# B&R Automation Studio project TD52 (part 61)

```c
  /* Logic: '<S427>/Logical Operator11' incorporates:
   *  Logic: '<S427>/Logical Operator25'
   *  UnitDelay: '<S427>/Unit Delay4'
   */
  rtb_LogicalOperator_in = ((!Gen2_ref_DWork->TOF_state) &&
    rtb_LogicalOperator5_mv && rtb_dbg_HLCi &&
    Gen2_ref_B->BusInput3.LR.bP_LoadReject_Active && rtb_RelationalOperator2_j);

  /* Sum: '<S427>/Sum6' incorporates:
   *  Constant: '<S427>/Constant7'
   *  Gain: '<S427>/Gain3'
   */
  rtb_Divide4_ia = 0.001 * Gen2_ref_B->BusInput3.LR.rTi_LR_GasStop + 0.01;

  /* Outputs for Atomic SubSystem: '<S427>/TOF1' */
  Gen2_ref_TOF(rtb_LogicalOperator_in, rtb_Divide4_ia, &Gen2_ref_B->TOF1_o,
               &Gen2_ref_DWork->TOF1_o, inst);

  /* End of Outputs for SubSystem: '<S427>/TOF1' */

  /* Outputs for Atomic SubSystem: '<S427>/TP' */
  Gen2_ref_TP(rtb_LogicalOperator_in, rtb_Divide4_ia, &Gen2_ref_B->TP_p,
              &Gen2_ref_DWork->TP_p, inst);

  /* End of Outputs for SubSystem: '<S427>/TP' */

  /* Switch: '<S427>/Switch1' */
  if (Gen2_ref_B->BusInput3.LR.bTiTOF_GasSTop) {
    rtb_TOF_IN = Gen2_ref_B->TOF1_o.LogicalOperator1;
  } else {
    rtb_TOF_IN = Gen2_ref_B->TP_p.LogicalOperator1;
  }

  /* End of Switch: '<S427>/Switch1' */

  /* Switch: '<Root>/GasStop1' */
  rtb_dbg_HLCi = ((!rtb_LogicalOperator) && rtb_TOF_IN);

  /* Outputs for Atomic SubSystem: '<S8>/BDC_Trajectory' */
  /* Gain: '<S345>/Gain8' incorporates:
   *  Gain: '<S417>/Gain8'
   *  Gain: '<S760>/Gain8'
   */
  rtb_Switch_ct_tmp = 100000.0 * Gen2_ref_B->BusInput3.traj.rPr_p2s_Sr_Man;

  /* Product: '<S413>/delta rise limit' incorporates:
   *  Gain: '<S345>/Gain8'
   *  Product: '<S434>/delta rise limit'
   *  Product: '<S795>/delta rise limit'
   *  SampleTimeMath: '<S413>/sample time'
   *
   * About '<S413>/sample time':
   *  y = K where K = ( w * Ts )
   */
  rtb_Divide_mr_tmp_0 = rtb_Switch_ct_tmp * 0.01;

  /* End of Outputs for SubSystem: '<S8>/BDC_Trajectory' */
  rtb_Divide_kp = rtb_Divide_mr_tmp_0;

  /* Gain: '<S4>/bar2Pa6' incorporates:
   *  DataTypeConversion: '<S4>/Data Type Conversion27'
   */
  rtb_bar2Pa6 = 100000.0 * Gen2_ref_B->BusInput.rPr_p2sMan;

  /* Logic: '<S4>/Logical Operator3' incorporates:
   *  Logic: '<S4>/Logical Operator2'
   */
  rtb_LogicalOperator_in = ((!rtb_LogicalOperator) || rtb_bResetBdc);

  /* DiscreteIntegrator: '<S345>/Discrete-Time Integrator' */
  if (rtb_LogicalOperator_in || (Gen2_ref_DWork->DiscreteTimeIntegrator_PrevRese
       != 0)) {
    Gen2_ref_DWork->DiscreteTimeIntegrator_DSTATE = 1.0;
  }

  if (Gen2_ref_DWork->DiscreteTimeIntegrator_DSTATE >= 1.0) {
    Gen2_ref_DWork->DiscreteTimeIntegrator_DSTATE = 1.0;
  } else if (Gen2_ref_DWork->DiscreteTimeIntegrator_DSTATE <= 0.0) {
    Gen2_ref_DWork->DiscreteTimeIntegrator_DSTATE = 0.0;
  }

  /* Logic: '<S345>/Logical Operator' incorporates:
   *  Constant: '<S345>/Constant2'
   *  DiscreteIntegrator: '<S345>/Discrete-Time Integrator'
   *  RelationalOperator: '<S345>/Relational Operator'
   */
  rtb_LogicalOperator_cn = ((0.99 <=
    Gen2_ref_DWork->DiscreteTimeIntegrator_DSTATE) || rtb_LogicalOperator_in);

  /* Delay: '<S413>/Delay' */
  Gen2_ref_DWork->icLoad_n = ((((Gen2_ref_PrevZCSigState->Delay_Reset_ZCE_k == 1)
    != (int32_T)rtb_LogicalOperator_cn) &&
    (Gen2_ref_PrevZCSigState->Delay_Reset_ZCE_k != 3)) || rtb_LogicalOperator_cn
    || Gen2_ref_DWork->icLoad_n);
  Gen2_ref_PrevZCSigState->Delay_Reset_ZCE_k = rtb_LogicalOperator_cn;
  if (Gen2_ref_DWork->icLoad_n) {
    Gen2_ref_DWork->Delay_DSTATE_n = rtb_bar2Pa6;
  }

  /* Sum: '<S413>/Difference Inputs1' incorporates:
   *  Delay: '<S413>/Delay'
   *  Switch: '<S413>/etaVolConst'
   */
  rtb_Divide4_ia = rtb_bar2Pa6 - Gen2_ref_DWork->Delay_DSTATE_n;

  /* Switch: '<S416>/Switch2' incorporates:
   *  Product: '<S413>/delta rise limit'
   *  RelationalOperator: '<S416>/LowerRelop1'
   */
  if (!(rtb_Divide4_ia > rtb_Divide_mr_tmp_0)) {
    /* Product: '<S413>/delta fall limit' incorporates:
     *  Gain: '<S345>/Gain15'
     *  Gain: '<S345>/Gain8'
     *  SampleTimeMath: '<S413>/sample time'
     *
     * About '<S413>/sample time':
     *  y = K where K = ( w * Ts )
     */
    rtb_Switch_ed = -rtb_Switch_ct_tmp * 0.01;

    /* Switch: '<S416>/Switch' incorporates:
     *  RelationalOperator: '<S416>/UpperRelop'
     */
    if (rtb_Divide4_ia < rtb_Switch_ed) {
      rtb_Divide_kp = rtb_Switch_ed;
    } else {
      rtb_Divide_kp = rtb_Divide4_ia;
    }

    /* End of Switch: '<S416>/Switch' */
  }

  /* End of Switch: '<S416>/Switch2' */

  /* Sum: '<S413>/Difference Inputs2' incorporates:
   *  Delay: '<S413>/Delay'
   */
  rtb_Divide4_ia = rtb_Divide_kp + Gen2_ref_DWork->Delay_DSTATE_n;

  /* Outputs for Atomic SubSystem: '<S345>/p2sfilt' */
  Gen2_ref_N_TC_HP_filt(rtb_Divide4_ia,
                        Gen2_ref_B->BusInput3.traj.rTiF_Pr_p2s_Man,
                        rtb_LogicalOperator_cn, &Gen2_ref_B->p2sfilt,
                        &Gen2_ref_DWork->p2sfilt, inst);

  /* End of Outputs for SubSystem: '<S345>/p2sfilt' */

  /* Gain: '<S875>/kW2W1' incorporates:
   *  Gain: '<S343>/Pa2bar2'
   *  Gain: '<S344>/kW2W1'
   *  Gain: '<S586>/Gain1'
   *  Gain: '<S639>/kW2W'
   *  Gain: '<S761>/kW2W'
   *  Switch: '<S761>/Switch2'
   */
  rtb_Product1_aq = 1000.0 * Gen2_ref_B->BusInput3.eng.rP_Nom;

  /* Product: '<S881>/delta rise limit' incorporates:
   *  Gain: '<S875>/kW2W1'
   *  Product: '<S875>/Divide1'
   *  SampleTimeMath: '<S881>/sample time'
   *
   * About '<S881>/sample time':
   *  y = K where K = ( w * Ts )
   */
  rtb_Divide2_a = rtb_Product1_aq *
    Gen2_ref_B->BusInput3.traj.rP_Ramp_IncGrad_Norm * 0.01;

  /* Product: '<S875>/Product' incorporates:
   *  Gain: '<S875>/kW2W1'
   */
  rtb_Product_gj = rtb_Product1_aq * Gen2_ref_B->BusInput3.eng.rP_Start_Norm;

  /* Outputs for Atomic SubSystem: '<S194>/Pel_filt' */
  Gen2_ref_N_TC_HP_filt(rtb_Gain2_ao, Gen2_ref_B->BusInput3.inFilt.rTiF_P,
                        rtb_bResetBdc, &Gen2_ref_B->Pel_filt,
                        &Gen2_ref_DWork->Pel_filt, inst);

  /* End of Outputs for SubSystem: '<S194>/Pel_filt' */

  /* MATLAB Function: '<S874>/MATLAB Function' */
  if (!Gen2_ref_B->BusInput.tLvrt.bLvrtFlg) {
    rtb_PactOut = Gen2_ref_B->Pel_filt.Switch;
    rtb_PrefOut = rtb_kW2W;
    Gen2_ref_DWork->LVRTFlgRise = false;
  } else if (Gen2_ref_B->BusInput.tLvrt.bLvrtFlg &&
             (!Gen2_ref_DWork->LVRTFlgRise)) {
    Gen2_ref_DWork->PFix = Gen2_ref_B->Pel_filt.Switch;
    rtb_PactOut = Gen2_ref_DWork->PFix;
    rtb_PrefOut = Gen2_ref_DWork->PFix;
    Gen2_ref_DWork->LVRTFlgRise = true;
  } else {
    rtb_PactOut = Gen2_ref_DWork->PFix;
    rtb_PrefOut = Gen2_ref_DWork->PFix;
  }

  /* End of MATLAB Function: '<S874>/MATLAB Function' */

  /* Switch: '<S881>/etaVolConst' incorporates:
   *  Constant: '<S875>/ tde2'
   *  Gain: '<S875>/kW2W1'
   *  RelationalOperator: '<S878>/LowerRelop1'
   *  RelationalOperator: '<S878>/UpperRelop'
   *  Switch: '<S878>/Switch'
   *  Switch: '<S878>/Switch2'
   */
  if (Gen2_ref_B->BusInput.bResetTraj) {
    rtb_PactOut = rtb_Product_gj;
  } else {
    if (rtb_PrefOut > rtb_Product1_aq) {
      /* Switch: '<S878>/Switch2' incorporates:
       *  Gain: '<S875>/kW2W1'
       */
      rtb_PrefOut = rtb_Product1_aq;
    } else if (rtb_PrefOut < 1.0) {
      /* Switch: '<S878>/Switch' incorporates:
       *  Constant: '<S875>/ tde2'
       *  Switch: '<S878>/Switch2'
       */
      rtb_PrefOut = 1.0;
    }

    /* Switch: '<S880>/Switch2' incorporates:
     *  Constant: '<S875>/ tde2'
     *  Gain: '<S875>/kW2W1'
     *  RelationalOperator: '<S878>/UpperRelop'
     *  RelationalOperator: '<S880>/LowerRelop1'
     *  RelationalOperator: '<S880>/UpperRelop'
     *  Switch: '<S878>/Switch'
     *  Switch: '<S878>/Switch2'
     *  Switch: '<S880>/Switch'
     */
    if (rtb_PactOut > rtb_Product1_aq) {
      rtb_PactOut = rtb_Product1_aq;
    } else if (rtb_PactOut < rtb_Product_gj) {
      /* Switch: '<S880>/Switch' */
      rtb_PactOut = rtb_Product_gj;
    }

    /* End of Switch: '<S880>/Switch2' */

    /* Sum: '<S875>/Sum10' incorporates:
     *  Gain: '<S875>/kW2W1'
     *  Product: '<S875>/Divide5'
     */
    rtb_PactOut += Gen2_ref_B->BusInput3.traj.rP_Diff_Max_Norm * rtb_Product1_aq;

    /* Switch: '<S879>/Switch2' incorporates:
     *  RelationalOperator: '<S879>/LowerRelop1'
     */
    if (!(rtb_PrefOut > rtb_PactOut)) {
      /* Switch: '<S879>/Switch' incorporates:
       *  Constant: '<S875>/ tde3'
       *  RelationalOperator: '<S879>/UpperRelop'
       */
      if (rtb_PrefOut < 1.0) {
        rtb_PactOut = 1.0;
      } else {
        rtb_PactOut = rtb_PrefOut;
      }

      /* End of Switch: '<S879>/Switch' */
    }

    /* End of Switch: '<S879>/Switch2' */
  }

  /* End of Switch: '<S881>/etaVolConst' */

  /* Delay: '<S881>/Delay' */
  Gen2_ref_DWork->icLoad_m = ((((Gen2_ref_PrevZCSigState->Delay_Reset_ZCE_b == 1)
    != (int32_T)Gen2_ref_B->BusInput.bResetTraj) &&
    (Gen2_ref_PrevZCSigState->Delay_Reset_ZCE_b != 3)) ||
    Gen2_ref_B->BusInput.bResetTraj || Gen2_ref_DWork->icLoad_m);
  Gen2_ref_PrevZCSigState->Delay_Reset_ZCE_b = Gen2_ref_B->BusInput.bResetTraj;
  if (Gen2_ref_DWork->icLoad_m) {
    Gen2_ref_DWork->Delay_DSTATE_oh = rtb_Product_gj;
  }

  /* Sum: '<S881>/Difference Inputs1' incorporates:
   *  Delay: '<S881>/Delay'
   */
  rtb_PactOut -= Gen2_ref_DWork->Delay_DSTATE_oh;

  /* Switch: '<S884>/Switch2' incorporates:
   *  RelationalOperator: '<S884>/LowerRelop1'
   */
  if (!(rtb_PactOut > rtb_Divide2_a)) {
    /* Product: '<S881>/delta fall limit' incorporates:
     *  Abs: '<S875>/Abs2'
     *  Gain: '<S875>/Gain2'
     *  Gain: '<S875>/kW2W1'
     *  Product: '<S875>/Divide2'
     *  SampleTimeMath: '<S881>/sample time'
     *
     * About '<S881>/sample time':
     *  y = K where K = ( w * Ts )
     */
    rtb_Switch_ed = -fabs(rtb_Product1_aq *
                          Gen2_ref_B->BusInput3.traj.rP_Ramp_DecGrad_Norm) *
      0.01;

    /* Switch: '<S884>/Switch' incorporates:
     *  RelationalOperator: '<S884>/UpperRelop'
     */
    if (rtb_PactOut < rtb_Switch_ed) {
      rtb_Divide2_a = rtb_Switch_ed;
    } else {
      rtb_Divide2_a = rtb_PactOut;
    }

    /* End of Switch: '<S884>/Switch' */
  }

  /* End of Switch: '<S884>/Switch2' */

  /* Sum: '<S881>/Difference Inputs2' incorporates:
   *  Delay: '<S881>/Delay'
   */
  rtb_Switch_ed = rtb_Divide2_a + Gen2_ref_DWork->Delay_DSTATE_oh;

  /* Outputs for Atomic SubSystem: '<S875>/Pd_filt' */
  Gen2_ref_Pd_filt(rtb_Switch_ed, Gen2_ref_B->BusInput3.traj.rTiFpowtraj,
                   rtb_Product_gj, Gen2_ref_B->BusInput.bResetTraj,
                   &Gen2_ref_B->Pd_filt_p, &Gen2_ref_DWork->Pd_filt_p, inst);

  /* End of Outputs for SubSystem: '<S875>/Pd_filt' */

  /* Gain: '<S344>/kW2W1' */
  rtb_kW2W1_h = rtb_Product1_aq;

  /* Product: '<S404>/delta rise limit' incorporates:
   *  Product: '<S344>/Divide1'
   *  SampleTimeMath: '<S404>/sample time'
   *
   * About '<S404>/sample time':
   *  y = K where K = ( w * Ts )
   */
  rtb_Divide2_a = rtb_kW2W1_h * Gen2_ref_B->BusInput3.traj.rP_Ramp_IncGrad_Norm *
    0.01;

  /* Product: '<S344>/Product' */
  rtb_PactOut = rtb_kW2W1_h * Gen2_ref_B->BusInput3.eng.rP_Start_Norm;

  /* Logic: '<Root>/Logical Operator1' incorporates:
   *  Logic: '<Root>/Logical Operator2'
   */
  rtb_LogicalOperator1_e = (Gen2_ref_B->BusInput.tLvrt.bLvrtFlg &&
    (!rtb_LogicalOperator_in));

  /* MATLAB Function: '<S339>/MATLAB Function' */
  if (!rtb_LogicalOperator1_e) {
    rtb_PactOut_o = Gen2_ref_B->Pel_filt.Switch;
    rtb_Product_gj = rtb_kW2W;
    Gen2_ref_DWork->LVRTFlgRise_e = false;
  } else if (!Gen2_ref_DWork->LVRTFlgRise_e) {
    Gen2_ref_DWork->PFix_g = Gen2_ref_B->Pel_filt.Switch;
    rtb_PactOut_o = Gen2_ref_DWork->PFix_g;
    rtb_Product_gj = Gen2_ref_DWork->PFix_g;
    Gen2_ref_DWork->LVRTFlgRise_e = true;
  } else {
    rtb_PactOut_o = Gen2_ref_DWork->PFix_g;
    rtb_Product_gj = Gen2_ref_DWork->PFix_g;
  }

  /* End of MATLAB Function: '<S339>/MATLAB Function' */

  /* Switch: '<S397>/Switch2' incorporates:
   *  Constant: '<S344>/ tde2'
   *  RelationalOperator: '<S397>/LowerRelop1'
   *  RelationalOperator: '<S397>/UpperRelop'
   *  Switch: '<S397>/Switch'
   */
  if (rtb_Product_gj > rtb_kW2W1_h) {
    rtb_PrefOut = rtb_kW2W1_h;
  } else if (rtb_Product_gj < 1.0) {
    /* Switch: '<S397>/Switch' incorporates:
     *  Constant: '<S344>/ tde2'
     */
    rtb_PrefOut = 1.0;
  } else {
    rtb_PrefOut = rtb_Product_gj;
  }

  /* End of Switch: '<S397>/Switch2' */

  /* Switch: '<S404>/etaVolConst' incorporates:
   *  RelationalOperator: '<S399>/LowerRelop1'
   *  RelationalOperator: '<S399>/UpperRelop'
   *  Switch: '<S399>/Switch'
   *  Switch: '<S399>/Switch2'
   */
  if (rtb_LogicalOperator_in) {
    rtb_Product_gj = rtb_PactOut;
  } else {
    if (rtb_PactOut_o > rtb_kW2W1_h) {
      /* Switch: '<S399>/Switch2' */
      rtb_Divide_kp = rtb_kW2W1_h;
    } else if (rtb_PactOut_o < rtb_PactOut) {
      /* Switch: '<S399>/Switch' incorporates:
       *  Switch: '<S399>/Switch2'
       */
      rtb_Divide_kp = rtb_PactOut;
    } else {
      /* Switch: '<S399>/Switch2' incorporates:
       *  Switch: '<S399>/Switch'
       */
      rtb_Divide_kp = rtb_PactOut_o;
    }

    /* Sum: '<S344>/Sum10' incorporates:
     *  Product: '<S344>/Divide5'
     *  RelationalOperator: '<S399>/UpperRelop'
     *  Switch: '<S399>/Switch'
     *  Switch: '<S399>/Switch2'
     */
    rtb_Product_gj = Gen2_ref_B->BusInput3.traj.rP_Diff_Max_Norm * rtb_kW2W1_h +
      rtb_Divide_kp;

    /* Switch: '<S398>/Switch2' incorporates:
     *  RelationalOperator: '<S398>/LowerRelop1'
     */
    if (!(rtb_PrefOut > rtb_Product_gj)) {
      /* Switch: '<S398>/Switch' incorporates:
       *  Constant: '<S344>/ tde3'
       *  RelationalOperator: '<S398>/UpperRelop'
       */
      if (rtb_PrefOut < 1.0) {
        rtb_Product_gj = 1.0;
      } else {
        rtb_Product_gj = rtb_PrefOut;
      }

      /* End of Switch: '<S398>/Switch' */
    }

    /* End of Switch: '<S398>/Switch2' */
  }

  /* End of Switch: '<S404>/etaVolConst' */

  /* Delay: '<S404>/Delay' */
  Gen2_ref_DWork->icLoad_k = ((((Gen2_ref_PrevZCSigState->Delay_Reset_ZCE_n == 1)
    != (int32_T)rtb_LogicalOperator_in) &&
    (Gen2_ref_PrevZCSigState->Delay_Reset_ZCE_n != 3)) || rtb_LogicalOperator_in
    || Gen2_ref_DWork->icLoad_k);
  Gen2_ref_PrevZCSigState->Delay_Reset_ZCE_n = rtb_LogicalOperator_in;
  if (Gen2_ref_DWork->icLoad_k) {
    Gen2_ref_DWork->Delay_DSTATE_g = rtb_PactOut;
  }

  /* Sum: '<S404>/Difference Inputs1' incorporates:
   *  Delay: '<S404>/Delay'
   */
  rtb_Product_gj -= Gen2_ref_DWork->Delay_DSTATE_g;

  /* Switch: '<S411>/Switch2' incorporates:
   *  RelationalOperator: '<S411>/LowerRelop1'
   */
  if (!(rtb_Product_gj > rtb_Divide2_a)) {
    /* Product: '<S404>/delta fall limit' incorporates:
     *  Abs: '<S344>/Abs2'
     *  Gain: '<S344>/Gain2'
     *  Product: '<S344>/Divide2'
     *  SampleTimeMath: '<S404>/sample time'
     *
     * About '<S404>/sample time':
     *  y = K where K = ( w * Ts )
     */
    rtb_deltafalllimit_ca = -fabs(rtb_kW2W1_h *
      Gen2_ref_B->BusInput3.traj.rP_Ramp_DecGrad_Norm) * 0.01;

    /* Switch: '<S411>/Switch' incorporates:
     *  RelationalOperator: '<S411>/UpperRelop'
     */
    if (rtb_Product_gj < rtb_deltafalllimit_ca) {
      rtb_Divide2_a = rtb_deltafalllimit_ca;
    } else {
      rtb_Divide2_a = rtb_Product_gj;
    }

    /* End of Switch: '<S411>/Switch' */
  }

  /* End of Switch: '<S411>/Switch2' */

  /* Sum: '<S404>/Difference Inputs2' incorporates:
   *  Delay: '<S404>/Delay'
   */
  rtb_Product_gj = rtb_Divide2_a + Gen2_ref_DWork->Delay_DSTATE_g;

  /* Outputs for Atomic SubSystem: '<S344>/Pd_filt' */
  Gen2_ref_Pd_filt(rtb_Product_gj, Gen2_ref_B->BusInput3.traj.rTiFpowtraj,
                   rtb_PactOut, rtb_LogicalOperator_in, &Gen2_ref_B->Pd_filt,
                   &Gen2_ref_DWork->Pd_filt, inst);

  /* End of Outputs for SubSystem: '<S344>/Pd_filt' */

  /* Gain: '<S344>/kW2W2' */
  rtb_PactOut = 1000.0 * rtb_kW2W1_h;

  /* Gain: '<S344>/kW2W3' */
  rtb_Divide2_a = 0.1 * rtb_PactOut;

  /* Outputs for Atomic SubSystem: '<S344>/WO1' */
  Gen2_ref_Filter1(rtb_PrefOut, Gen2_ref_B->BusInput3.traj.rTi_FSM_WO_1,
                   rtb_LogicalOperator_in, &Gen2_ref_B->WO1,
                   &Gen2_ref_DWork->WO1, inst);

  /* End of Outputs for SubSystem: '<S344>/WO1' */

  /* Outputs for Atomic SubSystem: '<S344>/WO2' */
  Gen2_ref_Filter3(Gen2_ref_B->WO1.Switch1,
                   Gen2_ref_B->BusInput3.traj.rTi_FSM_WO_2, Gen2_ref_ConstB.tde1,
                   rtb_LogicalOperator_in, &Gen2_ref_B->WO2,
                   &Gen2_ref_DWork->WO2, inst);

  /* End of Outputs for SubSystem: '<S344>/WO2' */

  /* Product: '<S344>/Divide3' */
  rtb_PrefOut = Gen2_ref_B->BusInput3.traj.rK_FSM_WO * Gen2_ref_B->WO2.Switch;

  /* Switch: '<S400>/Switch2' incorporates:
   *  RelationalOperator: '<S400>/LowerRelop1'
   */
  if (rtb_PrefOut > rtb_Divide2_a) {
    rtb_Switch2_g3 = rtb_Divide2_a;
  } else {
    /* Gain: '<S344>/kW2W4' */
    rtb_PactOut *= -0.1;

    /* Switch: '<S400>/Switch' incorporates:
     *  RelationalOperator: '<S400>/UpperRelop'
     */
    if (rtb_PrefOut < rtb_PactOut) {
      rtb_Switch2_g3 = rtb_PactOut;
    } else {
      rtb_Switch2_g3 = rtb_PrefOut;
    }

    /* End of Switch: '<S400>/Switch' */
  }

  /* End of Switch: '<S400>/Switch2' */

  /* Switch: '<S7>/Switch1' */
  if (Gen2_ref_B->BusInput3.traj.bUseSpeedCtrlPd) {
    rtb_kW2W1_h = Gen2_ref_B->Pd_filt_p.Switch;
  } else {
    /* Sum: '<S344>/Sum1' */
    rtb_PactOut = Gen2_ref_B->Pd_filt.Switch + rtb_Switch2_g3;

    /* Switch: '<S401>/Switch2' incorporates:
     *  RelationalOperator: '<S401>/LowerRelop1'
     */
    if (!(rtb_PactOut > rtb_kW2W1_h)) {
      /* Switch: '<S401>/Switch' incorporates:
       *  Constant: '<S344>/ tde4'
       *  RelationalOperator: '<S401>/UpperRelop'
       */
      if (rtb_PactOut < 1.0) {
        rtb_kW2W1_h = 1.0;
      } else {
        rtb_kW2W1_h = rtb_PactOut;
      }

      /* End of Switch: '<S401>/Switch' */
    }

    /* End of Switch: '<S401>/Switch2' */
  }

  /* End of Switch: '<S7>/Switch1' */

  /* Gain: '<S338>/W2kW' incorporates:
   *  Gain: '<S16>/W2kW'
   */
  rtb_PactOut_tmp = 0.001 * rtb_kW2W1_h;

  /* Switch: '<S376>/Switch2' incorporates:
   *  Gain: '<S338>/W2kW'
   *  RelationalOperator: '<S376>/LowerRelop1'
   */
  if (rtb_PactOut_tmp > Gen2_ref_B->BusInput3.eng.rP_Nom) {
    rtb_PrefOut = Gen2_ref_B->BusInput3.eng.rP_Nom;
  } else {
    /* Product: '<S373>/Divide6' */
    rtb_PrefOut = Gen2_ref_B->BusInput3.eng.rP_Nom *
      Gen2_ref_B->BusInput3.leanox.rP_P2sRedIP_SP_Norm;

    /* Switch: '<S376>/Switch' incorporates:
     *  RelationalOperator: '<S376>/UpperRelop'
     */
    if (!(rtb_PactOut_tmp < rtb_PrefOut)) {
      rtb_PrefOut = rtb_PactOut_tmp;
    }

    /* End of Switch: '<S376>/Switch' */
  }

  /* End of Switch: '<S376>/Switch2' */

  /* MATLAB Function: '<S373>/2-point interpolation, with extrapolation' */
  upointinterpolationwithextrapol(rtb_PrefOut,
    Gen2_ref_B->BusInput3.leanox.Comp_IgnP_x,
    Gen2_ref_B->BusInput3.leanox.Comp_IgnP_y,
    &Gen2_ref_B->sf_2pointinterpolationwithextra, inst);

  /* Outputs for Atomic SubSystem: '<S190>/N_TC_HP_filt' */
  /* DataTypeConversion: '<S4>/Data Type Conversion14' */
  Gen2_ref_N_TC_HP_filt((real_T)Gen2_ref_B->BusInput.rCA_Ign_Avg,
                        Gen2_ref_B->BusInput3.inFilt.rTiF_Ign, rtb_bResetBdc,
                        &Gen2_ref_B->N_TC_HP_filt, &Gen2_ref_DWork->N_TC_HP_filt, inst);

  /* End of Outputs for SubSystem: '<S190>/N_TC_HP_filt' */

  /* Switch: '<S377>/Switch2' incorporates:
   *  Gain: '<S338>/W2kW'
   *  RelationalOperator: '<S377>/LowerRelop1'
   */
  if (rtb_PactOut_tmp > Gen2_ref_B->BusInput3.eng.rP_Nom) {
    rtb_PrefOut = Gen2_ref_B->BusInput3.eng.rP_Nom;
  } else {
    /* Product: '<S373>/Divide1' */
    rtb_PrefOut = Gen2_ref_B->BusInput3.eng.rP_Nom *
      Gen2_ref_B->BusInput3.leanox.rP2s_Comp_Act_SP;

    /* Switch: '<S377>/Switch' incorporates:
     *  RelationalOperator: '<S377>/UpperRelop'
     */
    if (!(rtb_PactOut_tmp < rtb_PrefOut)) {
      rtb_PrefOut = rtb_PactOut_tmp;
    }

    /* End of Switch: '<S377>/Switch' */
  }

  /* End of Switch: '<S377>/Switch2' */

  /* MATLAB Function: '<S373>/2-point interpolation, with extrapolation1' */
  upointinterpolationwithextrapol(rtb_PrefOut,
    Gen2_ref_B->BusInput3.leanox.Comp_ChTmp_x,
    Gen2_ref_B->BusInput3.leanox.Comp_ChTmp_y,
    &Gen2_ref_B->sf_2pointinterpolationwithext_d, inst);

  /* Outputs for Atomic SubSystem: '<S197>/T2s_filt' */
  /* Bias: '<S4>/C2K2' incorporates:
   *  DataTypeConversion: '<S4>/Data Type Conversion9'
   */
  Gen2_ref_N_TC_HP_filt(Gen2_ref_B->BusInput.tT.rT2s + 273.15,
                        Gen2_ref_B->BusInput3.inFilt.rTiF_T, rtb_bResetBdc,
                        &Gen2_ref_B->T2s_filt, &Gen2_ref_DWork->T2s_filt, inst);

  /* End of Outputs for SubSystem: '<S197>/T2s_filt' */

  /* Switch: '<S338>/Switch1' incorporates:
   *  Gain: '<S338>/W2kW'
   *  Product: '<S338>/Divide6'
   *  Sum: '<S338>/Add4'
   */
  if (Gen2_ref_B->BusInput.tLEANOXin.bZylAusfall) {
    /* Switch: '<S355>/Switch' incorporates:
     *  Abs: '<S355>/Abs'
     *  Constant: '<S355>/Constant2'
     *  RelationalOperator: '<S355>/Relational Operator'
     */
    if (1.0 >= fabs(Gen2_ref_B->BusInput3.eng.rNum_Cyl_Eng)) {
      rtb_bResetHlci_0 = 1.0;
    } else {
      rtb_bResetHlci_0 = Gen2_ref_B->BusInput3.eng.rNum_Cyl_Eng;
    }

    /* End of Switch: '<S355>/Switch' */
    rtb_deltafalllimit_ca = rtb_PactOut_tmp / rtb_bResetHlci_0 + rtb_PactOut_tmp;
  } else {
    rtb_deltafalllimit_ca = rtb_PactOut_tmp;
  }

  /* End of Switch: '<S338>/Switch1' */

  /* Outputs for Atomic SubSystem: '<S193>/N_TC_LP_filt' */
  Gen2_ref_N_TC_HP_filt(rtb_DataTypeConversion15,
                        Gen2_ref_B->BusInput3.inFilt.rTiF_N, rtb_bResetBdc,
                        &Gen2_ref_B->N_TC_LP_filt_f,
                        &Gen2_ref_DWork->N_TC_LP_filt_f, inst);

  /* End of Outputs for SubSystem: '<S193>/N_TC_LP_filt' */

  /* Switch: '<S7>/Switch' */
  if (Gen2_ref_B->BusInput3.leanox.bMeasuredSpeed) {
    rtb_MinMax_n = Gen2_ref_B->N_TC_LP_filt_f.Switch;
  } else {
    rtb_MinMax_n = Gen2_ref_B->BusInput3.eng.rN_Nom;
  }

  /* End of Switch: '<S7>/Switch' */

  /* Switch: '<S346>/Switch' incorporates:
   *  Abs: '<S346>/Abs'
   *  Constant: '<S346>/Constant2'
   *  RelationalOperator: '<S346>/Relational Operator'
   */
  if (1.0 >= fabs(rtb_MinMax_n)) {
    rtb_Switch_on = 1.0;
  } else {
    rtb_Switch_on = rtb_MinMax_n;
  }

  /* End of Switch: '<S346>/Switch' */

  /* Switch: '<S338>/Switch4' */
  if (Gen2_ref_B->BusInput3.leanox.bLp_c_Ena) {
    rtb_bResetHlci_0 = Gen2_ref_B->BusInput3.leanox.rP_c;
  } else {
    rtb_bResetHlci_0 = Gen2_ref_B->BusInput3.leanox.rP_1;
  }

  /* End of Switch: '<S338>/Switch4' */

  /* Switch: '<S338>/Switch2' incorporates:
   *  Logic: '<S338>/Logical Operator1'
   *  Product: '<S338>/Divide4'
   *  RelationalOperator: '<S338>/Relational Operator1'
   *  RelationalOperator: '<S338>/Relational Operator3'
   *  Sum: '<S338>/Add5'
   *  Switch: '<S338>/Switch5'
   */
  if (rtb_deltafalllimit_ca < rtb_bResetHlci_0) {
    /* Switch: '<S338>/Switch_b_c' incorporates:
     *  Logic: '<S338>/Logical Operator'
     *  RelationalOperator: '<S338>/Relational Operator2'
     */
    if (Gen2_ref_B->BusInput3.leanox.bLp_c_Ena && (rtb_deltafalllimit_ca <
         Gen2_ref_B->BusInput3.leanox.rP_c)) {
      /* SignalConversion generated from: '<S338>/Lookup Table Dynamic1' */
      rtb_TmpSignalConversionAtLoo_ht[0] =
        Gen2_ref_B->BusInput3.leanox.rPr_mbar_0;

      /* Switch: '<S356>/Switch' incorporates:
       *  Abs: '<S356>/Abs'
       *  Constant: '<S356>/Constant2'
       *  RelationalOperator: '<S356>/Relational Operator'
       */
      if (1.0 >= fabs(Gen2_ref_B->BusInput3.leanox.rT_c)) {
        rtb_bResetHlci_0 = 1.0;
      } else {
        rtb_bResetHlci_0 = Gen2_ref_B->BusInput3.leanox.rT_c;
      }

      /* End of Switch: '<S356>/Switch' */

      /* SignalConversion generated from: '<S338>/Lookup Table Dynamic1' incorporates:
       *  Product: '<S338>/Divide5'
       */
      rtb_TmpSignalConversionAtLoo_ht[1] =
        Gen2_ref_B->BusInput3.leanox.rPr_mbar_c *
        Gen2_ref_B->BusInput3.leanox.rN_c / rtb_bResetHlci_0 *
        Gen2_ref_B->T2s_filt.Switch / rtb_Switch_on;

      /* SignalConversion generated from: '<S338>/Lookup Table Dynamic1' incorporates:
       *  Constant: '<S338>/Pel_a (kW)1'
       */
      rtb_TmpSignalConversionAtLook_d[0] = 0.0;
      rtb_TmpSignalConversionAtLook_d[1] = Gen2_ref_B->BusInput3.leanox.rP_c;

      /* S-Function (sfix_look1_dyn): '<S338>/Lookup Table Dynamic1' */
      /* Dynamic Look-Up Table Block: '<S338>/Lookup Table Dynamic1'
       * Input0  Data Type:  Floating Point real_T
       * Input1  Data Type:  Floating Point real_T
       * Input2  Data Type:  Floating Point real_T
       * Output0 Data Type:  Floating Point real_T
       * Lookup Method: Linear_Endpoint
       *
       */
      LookUp_real_T_real_T( &(rtb_LookupTableDynamic1_e),
                           &rtb_TmpSignalConversionAtLoo_ht[0],
                           rtb_deltafalllimit_ca,
                           &rtb_TmpSignalConversionAtLook_d[0], 1U, inst);
      rtb_MinMax_n = rtb_LookupTableDynamic1_e;
    } else {
      /* SignalConversion generated from: '<S338>/Lookup Table Dynamic' */
      rtb_TmpSignalConversionAtLoo_ht[0] =
        Gen2_ref_B->BusInput3.leanox.rPr_mbar_0;

      /* Switch: '<S354>/Switch' incorporates:
       *  Abs: '<S354>/Abs'
       *  Constant: '<S354>/Constant2'
       *  RelationalOperator: '<S354>/Relational Operator'
       */
      if (1.0 >= fabs(Gen2_ref_B->BusInput3.leanox.rT_1)) {
        rtb_bResetHlci_0 = 1.0;
      } else {
        rtb_bResetHlci_0 = Gen2_ref_B->BusInput3.leanox.rT_1;
      }

      /* End of Switch: '<S354>/Switch' */

      /* SignalConversion generated from: '<S338>/Lookup Table Dynamic' incorporates:
       *  Product: '<S338>/Divide1'
       */
      rtb_TmpSignalConversionAtLoo_ht[1] =
        Gen2_ref_B->BusInput3.leanox.rPr_mbar_1 *
        Gen2_ref_B->BusInput3.leanox.rN_1 / rtb_bResetHlci_0 *
        Gen2_ref_B->T2s_filt.Switch / rtb_Switch_on;

      /* SignalConversion generated from: '<S338>/Lookup Table Dynamic' incorporates:
       *  Constant: '<S338>/Pel_a (kW)3'
       */
      rtb_TmpSignalConversionAtLook_d[0] = 0.0;
      rtb_TmpSignalConversionAtLook_d[1] = Gen2_ref_B->BusInput3.leanox.rP_1;

      /* S-Function (sfix_look1_dyn): '<S338>/Lookup Table Dynamic' */
      /* Dynamic Look-Up Table Block: '<S338>/Lookup Table Dynamic'
       * Input0  Data Type:  Floating Point real_T
       * Input1  Data Type:  Floating Point real_T
       * Input2  Data Type:  Floating Point real_T
       * Output0 Data Type:  Floating Point real_T
       * Lookup Method: Linear_Endpoint
       *
       */
      LookUp_real_T_real_T( &(rtb_LookupTableDynamic_i),
                           &rtb_TmpSignalConversionAtLoo_ht[0],
                           rtb_deltafalllimit_ca,
                           &rtb_TmpSignalConversionAtLook_d[0], 1U, inst);
      rtb_MinMax_n = rtb_LookupTableDynamic_i;
    }

    /* End of Switch: '<S338>/Switch_b_c' */
  } else {
    if (Gen2_ref_B->BusInput3.leanox.bLp_c_Ena && (rtb_deltafalllimit_ca <
         Gen2_ref_B->BusInput3.leanox.rP_1)) {
      /* Sum: '<S338>/Add1' incorporates:
       *  Switch: '<S338>/Switch5'
       */
      rtb_Switch_jz = Gen2_ref_B->BusInput3.leanox.rP_1 -
        Gen2_ref_B->BusInput3.leanox.rP_c;

      /* Sum: '<S338>/Sum4' incorporates:
       *  Switch: '<S338>/Switch5'
       */
      rtb_Divide2_a = Gen2_ref_B->BusInput3.leanox.rP_c +
        Gen2_ref_B->BusInput3.leanox.rP_Eng_Frict;

      /* Switch: '<S349>/Switch' incorporates:
       *  Abs: '<S349>/Abs'
       *  Constant: '<S349>/Constant2'
       *  RelationalOperator: '<S349>/Relational Operator'
       *  Switch: '<S338>/Switch5'
       */
      if (1.0 >= fabs(rtb_Divide2_a)) {
        rtb_rKK2_k = 1.0;
      } else {
        rtb_rKK2_k = rtb_Divide2_a;
      }

      /* End of Switch: '<S349>/Switch' */

      /* Sum: '<S338>/Sum5' incorporates:
       *  Switch: '<S338>/Switch5'
       */
      rtb_Divide2_a = Gen2_ref_B->BusInput3.leanox.rP_1 +
        Gen2_ref_B->BusInput3.leanox.rP_Eng_Frict;

      /* Switch: '<S357>/Switch' incorporates:
       *  Abs: '<S357>/Abs'
       *  Constant: '<S357>/Constant2'
       *  RelationalOperator: '<S357>/Relational Operator'
       *  Switch: '<S338>/Switch5'
       */
      if (1.0 >= fabs(Gen2_ref_B->BusInput3.leanox.rT_1)) {
        rtb_bResetHlci_0 = 1.0;
      } else {
        rtb_bResetHlci_0 = Gen2_ref_B->BusInput3.leanox.rT_1;
      }

      /* End of Switch: '<S357>/Switch' */

      /* Switch: '<S348>/Switch' incorporates:
       *  Abs: '<S348>/Abs'
       *  Constant: '<S348>/Constant2'
       *  RelationalOperator: '<S348>/Relational Operator'
       *  Switch: '<S338>/Switch5'
       */
      if (1.0 >= fabs(rtb_Divide2_a)) {
        rtb_Divide2_a = 1.0;
      }

      /* End of Switch: '<S348>/Switch' */

      /* Product: '<S338>/rKK3' incorporates:
       *  Switch: '<S338>/Switch5'
       */
      rtb_Divide2_a = Gen2_ref_B->BusInput3.leanox.rPr_mbar_1 *
        Gen2_ref_B->BusInput3.leanox.rN_1 / rtb_bResetHlci_0 / rtb_Divide2_a;

      /* Switch: '<S350>/Switch' incorporates:
       *  Abs: '<S350>/Abs'
       *  Constant: '<S350>/Constant2'
       *  RelationalOperator: '<S350>/Relational Operator'
       *  Switch: '<S338>/Switch5'
       */
      if (1.0 >= fabs(Gen2_ref_B->BusInput3.leanox.rT_c)) {
        rtb_bResetHlci_0 = 1.0;
      } else {
        rtb_bResetHlci_0 = Gen2_ref_B->BusInput3.leanox.rT_c;
      }

      /* End of Switch: '<S350>/Switch' */

      /* Switch: '<S358>/Switch' incorporates:
       *  Abs: '<S358>/Abs'
       *  Constant: '<S358>/Constant2'
       *  RelationalOperator: '<S358>/Relational Operator'
       *  Switch: '<S338>/Switch5'
       */
      if (1.0 >= fabs(rtb_Switch_jz)) {
        rtb_Switch_jz = 1.0;
      }

      /* End of Switch: '<S358>/Switch' */

      /* Switch: '<S338>/Switch5' incorporates:
       *  Gain: '<S338>/W2kW'
       *  Product: '<S338>/Divide10'
       *  Product: '<S338>/Divide9'
       *  Product: '<S338>/rKK4'
       *  Sum: '<S338>/Add3'
       *  Sum: '<S338>/Sum6'
       *  Sum: '<S338>/Sum7'
       */
      rtb_PactOut = (rtb_Divide2_a - Gen2_ref_B->BusInput3.leanox.rPr_mbar_c *
                     Gen2_ref_B->BusInput3.leanox.rN_c / rtb_bResetHlci_0 /
                     rtb_rKK2_k) / rtb_Switch_jz * (rtb_PactOut_tmp -
        Gen2_ref_B->BusInput3.leanox.rP_1) + rtb_Divide2_a;
    } else {
      /* Sum: '<S338>/Add10' incorporates:
       *  Switch: '<S338>/Switch5'
       */
      rtb_Switch_jz = Gen2_ref_B->BusInput3.leanox.rP_2 -
        Gen2_ref_B->BusInput3.leanox.rP_1;

      /* Sum: '<S338>/Sum' incorporates:
       *  Switch: '<S338>/Switch5'
       */
      rtb_rKK2_k = Gen2_ref_B->BusInput3.leanox.rP_1 +
        Gen2_ref_B->BusInput3.leanox.rP_Eng_Frict;

      /* Sum: '<S338>/Sum1' incorporates:
       *  Switch: '<S338>/Switch5'
       */
      rtb_Divide2_a = Gen2_ref_B->BusInput3.leanox.rP_2 +
        Gen2_ref_B->BusInput3.leanox.rP_Eng_Frict;

      /* Switch: '<S347>/Switch' incorporates:
       *  Abs: '<S347>/Abs'
       *  Constant: '<S347>/Constant2'
       *  RelationalOperator: '<S347>/Relational Operator'
       *  Switch: '<S338>/Switch5'
       */
      if (1.0 >= fabs(Gen2_ref_B->BusInput3.leanox.rT_2)) {
        rtb_bResetHlci_0 = 1.0;
      } else {
        rtb_bResetHlci_0 = Gen2_ref_B->BusInput3.leanox.rT_2;
      }

      /* End of Switch: '<S347>/Switch' */

      /* Switch: '<S352>/Switch' incorporates:
       *  Abs: '<S352>/Abs'
       *  Constant: '<S352>/Constant2'
       *  RelationalOperator: '<S352>/Relational Operator'
       *  Switch: '<S338>/Switch5'
       */
      if (1.0 >= fabs(rtb_Divide2_a)) {
        rtb_Divide2_a = 1.0;
      }

      /* End of Switch: '<S352>/Switch' */

      /* Product: '<S338>/rKK1' incorporates:
       *  Switch: '<S338>/Switch5'
       */
      rtb_Divide2_a = Gen2_ref_B->BusInput3.leanox.rPr_mbar_2 *
        Gen2_ref_B->BusInput3.leanox.rN_2 / rtb_bResetHlci_0 / rtb_Divide2_a;

      /* Switch: '<S353>/Switch' incorporates:
       *  Abs: '<S353>/Abs'
       *  Constant: '<S353>/Constant2'
       *  RelationalOperator: '<S353>/Relational Operator'
       *  Switch: '<S338>/Switch5'
       */
      if (1.0 >= fabs(rtb_rKK2_k)) {
        rtb_rKK2_k = 1.0;
      }

      /* End of Switch: '<S353>/Switch' */

      /* Switch: '<S351>/Switch' incorporates:
       *  Abs: '<S351>/Abs'
       *  Constant: '<S351>/Constant2'
       *  RelationalOperator: '<S351>/Relational Operator'
       *  Switch: '<S338>/Switch5'
       */
      if (1.0 >= fabs(rtb_Switch_jz)) {
        rtb_Switch_jz = 1.0;
      }

      /* End of Switch: '<S351>/Switch' */

      /* Switch: '<S338>/Switch5' incorporates:
       *  Gain: '<S338>/W2kW'
       *  Product: '<S338>/Divide2'
       *  Product: '<S338>/Divide3'
       *  Product: '<S338>/rKK2'
       *  Sum: '<S338>/Add2'
       *  Sum: '<S338>/Sum2'
       *  Sum: '<S338>/Sum3'
       */
      rtb_PactOut = (rtb_Divide2_a - Gen2_ref_B->BusInput3.leanox.rPr_mbar_1 *
                     Gen2_ref_B->BusInput3.leanox.rN_1 /
                     Gen2_ref_B->BusInput3.leanox.rT_1 / rtb_rKK2_k) /
        rtb_Switch_jz * (rtb_PactOut_tmp - Gen2_ref_B->BusInput3.leanox.rP_2) +
        rtb_Divide2_a;
    }

    rtb_MinMax_n = rtb_PactOut * Gen2_ref_B->T2s_filt.Switch *
      (Gen2_ref_B->BusInput3.leanox.rP_Eng_Frict + rtb_deltafalllimit_ca) /
      rtb_Switch_on;
  }

  /* End of Switch: '<S338>/Switch2' */

  /* Product: '<S359>/Divide8' incorporates:
   *  DataTypeConversion: '<S359>/Data Type Conversion2'
   */
  rtb_PactOut = rtb_MinMax_n * Gen2_ref_B->BusInput.tLEANOXin.rLEANOX_fact_BC;

  /* Delay: '<S15>/Resettable Delay' incorporates:
   *  Constant: '<S15>/Pel_a (kW)2'
   */
  Gen2_ref_DWork->icLoad_nl =
    ((((Gen2_ref_PrevZCSigState->ResettableDelay_Reset_ZCE == 1) != (int32_T)
       rtb_bResetBdc) && (Gen2_ref_PrevZCSigState->ResettableDelay_Reset_ZCE !=
       3)) || rtb_bResetBdc || Gen2_ref_DWork->icLoad_nl);
  Gen2_ref_PrevZCSigState->ResettableDelay_Reset_ZCE = rtb_bResetBdc;
  if (Gen2_ref_DWork->icLoad_nl) {
    Gen2_ref_DWork->ResettableDelay_DSTATE = 0.0;
  }

  /* Sum: '<S888>/Sum1' incorporates:
   *  Sum: '<S589>/Sum1'
   */
  rtb_Divide_mr_tmp = Gen2_ref_B->BusInput3.SkipF.rP_1 -
    Gen2_ref_B->BusInput3.SkipF.rP_0;

  /* Abs: '<S901>/Abs' incorporates:
   *  Abs: '<S596>/Abs'
   *  Sum: '<S888>/Sum1'
   */
  rtb_Switch2_ba = fabs(rtb_Divide_mr_tmp);

  /* Switch: '<S901>/Switch' incorporates:
   *  Abs: '<S901>/Abs'
   *  Constant: '<S901>/Constant2'
   *  RelationalOperator: '<S901>/Relational Operator'
   *  Sum: '<S888>/Sum1'
   */
  if (2.2204460492503131E-16 >= rtb_Switch2_ba) {
    rtb_bResetHlci_0 = 2.2204460492503131E-16;
  } else {
    rtb_bResetHlci_0 = rtb_Divide_mr_tmp;
  }

  /* End of Switch: '<S901>/Switch' */

  /* Sum: '<S888>/Sum3' incorporates:
   *  Gain: '<S888>/Gain'
   *  Product: '<S888>/Divide'
   *  Product: '<S888>/Product'
   *  Sum: '<S888>/Sum'
   *  Sum: '<S888>/Sum2'
   */
  rtb_deltafalllimit_ca = Gen2_ref_B->BusInput3.SkipF.rNum_P0 - (0.001 *
    rtb_kW2W1_h - Gen2_ref_B->BusInput3.SkipF.rP_0) *
    (Gen2_ref_B->BusInput3.SkipF.rNum_P0 / rtb_bResetHlci_0);

  /* Switch: '<S902>/Switch2' incorporates:
   *  Constant: '<S888>/Constant1'
   *  RelationalOperator: '<S902>/LowerRelop1'
   *  RelationalOperator: '<S902>/UpperRelop'
   *  Switch: '<S902>/Switch'
   */
  if (rtb_deltafalllimit_ca > Gen2_ref_B->BusInput3.eng.rNum_Cyl_Eng) {
    rtb_deltafalllimit_ca = Gen2_ref_B->BusInput3.eng.rNum_Cyl_Eng;
  } else if (rtb_deltafalllimit_ca < 0.0) {
    /* Switch: '<S902>/Switch' incorporates:
     *  Constant: '<S888>/Constant1'
     */
    rtb_deltafalllimit_ca = 0.0;
  }

  /* End of Switch: '<S902>/Switch2' */

  /* Rounding: '<S888>/Rounding Function' */
  rtb_MinMax_n = rt_roundd_snf(rtb_deltafalllimit_ca, inst);

  /* MinMax: '<S19>/MinMax' */
  if ((Gen2_ref_B->BusInput.iN_Skip_Ext >= rtb_MinMax_n) || rtIsNaN(rtb_MinMax_n))
  {
    rtb_MinMax_n = Gen2_ref_B->BusInput.iN_Skip_Ext;
  }

  /* End of MinMax: '<S19>/MinMax' */

  /* Sum: '<S19>/Sum4' */
  rtb_deltafalllimit_ca = Gen2_ref_B->BusInput3.eng.rNum_Cyl_Eng - rtb_MinMax_n;

  /* Switch: '<S892>/Switch2' incorporates:
   *  RelationalOperator: '<S892>/LowerRelop1'
   *  RelationalOperator: '<S892>/UpperRelop'
   *  Switch: '<S892>/Switch'
   */
  if (rtb_deltafalllimit_ca > Gen2_ref_B->BusInput3.eng.rNum_Cyl_Eng) {
    rtb_deltafalllimit_ca = Gen2_ref_B->BusInput3.eng.rNum_Cyl_Eng;
  } else if (rtb_deltafalllimit_ca < 1.0) {
    /* Switch: '<S892>/Switch' */
    rtb_deltafalllimit_ca = 1.0;
  }

  /* End of Switch: '<S892>/Switch2' */

  /* Outputs for Atomic SubSystem: '<S19>/Filter1' */
  /* Product: '<S19>/Divide1' */
  Gen2_ref_Filter3(Gen2_ref_B->BusInput3.eng.rNum_Cyl_Eng /
                   rtb_deltafalllimit_ca, Gen2_ref_B->BusInput3.SkipF.rTiF_stat,
                   1.0, rtb_bResetBdc, &Gen2_ref_B->Filter1_l,
                   &Gen2_ref_DWork->Filter1_l, inst);

  /* End of Outputs for SubSystem: '<S19>/Filter1' */

  /* Switch: '<S19>/NSkip1' incorporates:
   *  Constant: '<S19>/Constant5'
   *  Logic: '<S19>/Logical Operator1'
   */
  if (!Gen2_ref_B->BusInput3.SkipF.bSF_ON) {
    u0 = 1.0;
  } else {
    u0 = Gen2_ref_B->Filter1_l.Switch;
  }

  /* End of Switch: '<S19>/NSkip1' */

  /* Switch: '<S373>/Switch1' incorporates:
   *  Constant: '<S373>/Pel_a (kW)1'
   *  DataTypeConversion: '<S4>/Data Type Conversion22'
   *  Product: '<S373>/Divide5'
   *  Sum: '<S373>/Add12'
   */
  if (Gen2_ref_B->BusInput3.leanox.bZZPKorr) {
    rtb_bResetHlci_0 = (Gen2_ref_B->BusInput.rCA_Ign_OP_Power -
                        Gen2_ref_B->N_TC_HP_filt.Switch) *
      Gen2_ref_B->sf_2pointinterpolationwithextra.y;
  } else {
    rtb_bResetHlci_0 = 0.0;
  }

  /* End of Switch: '<S373>/Switch1' */

  /* Switch: '<S373>/Switch2' incorporates:
   *  Constant: '<S373>/Pel_a (kW)2'
   *  Product: '<S373>/Divide9'
   *  Sum: '<S373>/Add13'
   */
  if (Gen2_ref_B->BusInput3.leanox.bt2Korr) {
    delta_y = (Gen2_ref_B->T2s_filt.Switch - Gen2_ref_B->BusInput3.leanox.rT_2) *
      Gen2_ref_B->sf_2pointinterpolationwithext_d.y;
  } else {
    delta_y = 0.0;
  }

  /* End of Switch: '<S373>/Switch2' */

  /* Switch: '<S373>/Switch3' incorporates:
   *  Constant: '<S373>/Pel_a (kW)3'
   */
  if (Gen2_ref_B->BusInput3.leanox.bHum_Act) {
    FILT_IN = Gen2_ref_B->BusInput3.leanox.rP2s_Comp_HumOffset;
  } else {
    FILT_IN = 0.0;
  }

  /* End of Switch: '<S373>/Switch3' */

  /* MinMax: '<S359>/MinMax' incorporates:
   *  MinMax: '<S775>/MinMax'
   */
  rtb_bCBV_min = !rtIsNaN(Gen2_ref_B->BusInput.tLEANOXin.rHiCtr_Leanox_Corr);
  if ((!(u0 >= Gen2_ref_B->BusInput.tLEANOXin.rHiCtr_Leanox_Corr)) &&
      rtb_bCBV_min) {
    u0 = Gen2_ref_B->BusInput.tLEANOXin.rHiCtr_Leanox_Corr;
  }

  /* End of MinMax: '<S359>/MinMax' */

  /* Gain: '<S359>/mbar2pa' incorporates:
   *  DataTypeConversion: '<S359>/Data Type Conversion'
   *  Delay: '<S15>/Resettable Delay'
   *  Product: '<S359>/Divide5'
   *  Sum: '<S359>/Add1'
   *  Sum: '<S359>/Add11'
   *  Sum: '<S359>/Add9'
   */
  rtb_Pa2bar_k = (((((rtb_bResetHlci_0 + delta_y) + FILT_IN) + rtb_PactOut) +
                   Gen2_ref_DWork->ResettableDelay_DSTATE) * u0 +
                  Gen2_ref_B->BusInput.tLEANOXin.rLEANOXoffset) * 100.0;

  /* Saturate: '<S388>/Saturation' */
  if (Gen2_ref_B->BusInput3.SpeedCtrl.rPosValvethrshAW > 1.0) {
    /* Saturate: '<S490>/Saturation' incorporates:
     *  Saturate: '<S18>/Saturation'
     *  Saturate: '<S752>/Saturation'
     *  Switch: '<S752>/Switch2'
     */
    rtb_PactOut = 1.0;
  } else if (Gen2_ref_B->BusInput3.SpeedCtrl.rPosValvethrshAW < 0.0) {
    /* Saturate: '<S490>/Saturation' incorporates:
     *  Saturate: '<S18>/Saturation'
     *  Saturate: '<S752>/Saturation'
     *  Switch: '<S752>/Switch2'
     */
    rtb_PactOut = 0.0;
  } else {
    /* Saturate: '<S490>/Saturation' incorporates:
     *  Saturate: '<S18>/Saturation'
     *  Saturate: '<S752>/Saturation'
     *  Switch: '<S752>/Switch2'
     */
    rtb_PactOut = Gen2_ref_B->BusInput3.SpeedCtrl.rPosValvethrshAW;
  }

  /* Sum: '<S388>/Sum1' incorporates:
   *  Saturate: '<S388>/Saturation'
   *  Sum: '<S752>/Sum1'
   *  Switch: '<S752>/Switch2'
   */
  rtb_Switch2_ejy_tmp_0 = Gen2_ref_B->BusInput3.bdcCbv.rPos_min + rtb_PactOut;
  rtb_Switch2_l = rtb_Switch2_ejy_tmp_0;

  /* RelationalOperator: '<S388>/Relational Operator' incorporates:
   *  Delay: '<Root>/Delay4'
   */
  rtb_LogicalOperator_cn = (Gen2_ref_DWork->Delay4_DSTATE <= rtb_Switch2_l);

  /* Delay: '<Root>/Delay3' */
  rtb_Switch_on = Gen2_ref_DWork->Delay3_DSTATE;

  /* Saturate: '<S388>/Saturation2' */
  if (Gen2_ref_B->BusInput3.bdcTv.rPos_max > 1.0) {
    /* Saturate: '<S752>/Saturation2' incorporates:
     *  Saturate: '<S18>/Saturation2'
     *  Switch: '<S752>/Switch2'
     */
    rtb_PrefOut = 1.0;
  } else if (Gen2_ref_B->BusInput3.bdcTv.rPos_max < 0.1) {
    /* Saturate: '<S752>/Saturation2' incorporates:
     *  Saturate: '<S18>/Saturation2'
     *  Switch: '<S752>/Switch2'
     */
    rtb_PrefOut = 0.1;
  } else {
    /* Saturate: '<S752>/Saturation2' incorporates:
     *  Saturate: '<S18>/Saturation2'
     *  Switch: '<S752>/Switch2'
     */
    rtb_PrefOut = Gen2_ref_B->BusInput3.bdcTv.rPos_max;
  }

  rtb_Switch2_l = rtb_PrefOut;

  /* End of Saturate: '<S388>/Saturation2' */

  /* Product: '<S388>/Divide1' */
  rtb_deltafalllimit_ca = rtb_Switch_on / rtb_Switch2_l;

  /* Sum: '<S388>/Sum' incorporates:
   *  Constant: '<S388>/Constant4'
   *  Saturate: '<S388>/Saturation'
   */
  rtb_Switch2_l = 1.0 - rtb_PactOut;

  /* RelationalOperator: '<S388>/Relational Operator1' */
  rtb_LogicalOperator5_mv = (rtb_deltafalllimit_ca >= rtb_Switch2_l);

  /* Logic: '<S388>/Logical Operator' */
  rtb_LogicalOperator2_p1 = (rtb_LogicalOperator_cn && rtb_LogicalOperator5_mv);

  /* Switch: '<S388>/Switch' incorporates:
   *  Constant: '<S388>/Constant'
   *  Constant: '<S388>/Constant1'
   */
  if (rtb_LogicalOperator2_p1) {
    rtb_mbar2pa_g = 0.0;
  } else {
    rtb_mbar2pa_g = 1.0E+6;
  }

  /* End of Switch: '<S388>/Switch' */

  /* Outputs for Atomic SubSystem: '<S6>/TOF' */
  /* Delay: '<Root>/Delay6' */
  Gen2_ref_TOF(Gen2_ref_DWork->Delay6_DSTATE,
               Gen2_ref_B->BusInput3.GQC.rTOF_DetSat, &Gen2_ref_B->TOF,
               &Gen2_ref_DWork->TOF, inst);

  /* End of Outputs for SubSystem: '<S6>/TOF' */

  /* Logic: '<Root>/Logical Operator' incorporates:
   *  Logic: '<Root>/Logical Operator4'
   */
  rtb_LogicalOperator_cn = (rtb_LogicalOperator_in && rtb_bResetHlci);

  /* Delay: '<Root>/Delay2' incorporates:
   *  Bias: '<Root>/Bias'
   *  Delay: '<Root>/Delay1'
   *  Logic: '<Root>/Logical Operator'
   */
  Gen2_ref_DWork->icLoad_e = ((((Gen2_ref_PrevZCSigState->Delay2_Reset_ZCE == 1)
    != (int32_T)rtb_LogicalOperator_cn) &&
    (Gen2_ref_PrevZCSigState->Delay2_Reset_ZCE != 3)) || rtb_LogicalOperator_cn ||
    Gen2_ref_DWork->icLoad_e);
  Gen2_ref_PrevZCSigState->Delay2_Reset_ZCE = rtb_LogicalOperator_cn;
  if (Gen2_ref_DWork->icLoad_e) {
    Gen2_ref_DWork->Delay2_DSTATE = Gen2_ref_DWork->Delay1_DSTATE[1] + 0.01;
  }

  /* Logic: '<S6>/Logical Operator2' incorporates:
   *  Abs: '<S6>/Abs2'
   *  Abs: '<S6>/Abs3'
   *  Delay: '<Root>/Delay1'
   *  Delay: '<Root>/Delay2'
   *  RelationalOperator: '<S6>/Relational Operator2'
   *  RelationalOperator: '<S6>/Relational Operator3'
   *  Sum: '<S6>/Sum2'
   *  Sum: '<S6>/Sum3'
   */
  rtb_LogicalOperator2_fy = ((fabs(Gen2_ref_DWork->Delay2_DSTATE -
    Gen2_ref_DWork->Delay1_DSTATE[0]) < Gen2_ref_B->BusInput3.GQC.rThrshLamSat) ||
    (fabs(Gen2_ref_DWork->Delay2_DSTATE - Gen2_ref_DWork->Delay1_DSTATE[1]) <
     Gen2_ref_B->BusInput3.GQC.rThrshLamSat));

  /* Outputs for Atomic SubSystem: '<S6>/TON' */
  Gen2_ref_TON_1(rtb_LogicalOperator2_fy, Gen2_ref_B->BusInput3.GQC.rTON_LamSat,
                 &Gen2_ref_B->TON, &Gen2_ref_DWork->TON, inst);

  /* End of Outputs for SubSystem: '<S6>/TON' */

  /* Switch: '<S6>/Switch3' incorporates:
   *  Constant: '<S6>/Constant8'
   *  Logic: '<S6>/Logical Operator'
   *  Logic: '<S6>/Logical Operator1'
   */
  if (Gen2_ref_B->BusInput3.GQC.bEnableFuncQGC) {
    rtb_bActGasQualImprov = ((!Gen2_ref_B->TOF.LogicalOperator1) &&
      Gen2_ref_B->TON.LogicalOperator3);
  } else {
    rtb_bActGasQualImprov = false;
  }

  /* End of Switch: '<S6>/Switch3' */

  /* Sum: '<S343>/Sum2' incorporates:
   *  Sum: '<S342>/Sum2'
   */
  u0 = rtb_kW2W1_h - rtb_PactOut_o;

  /* Product: '<S343>/Product' incorporates:
   *  DataTypeConversion: '<S343>/Data Type Conversion'
   *  Gain: '<S343>/Gain4'
   *  Sum: '<S343>/Sum2'
   */
  rtb_Switch_jz = u0 * 1.0E-6 * (real_T)rtb_bActGasQualImprov;

  /* Saturate: '<S388>/Saturation1' */
  if (Gen2_ref_B->BusInput3.bdcCbv.rPos_max > 1.0) {
    /* Saturate: '<S490>/Saturation1' incorporates:
     *  Saturate: '<S18>/Saturation1'
     */
    rtb_deltafalllimit_ca = 1.0;
  } else if (Gen2_ref_B->BusInput3.bdcCbv.rPos_max < 0.1) {
    /* Saturate: '<S490>/Saturation1' incorporates:
     *  Saturate: '<S18>/Saturation1'
     */
    rtb_deltafalllimit_ca = 0.1;
  } else {
    /* Saturate: '<S490>/Saturation1' incorporates:
     *  Saturate: '<S18>/Saturation1'
     */
    rtb_deltafalllimit_ca = Gen2_ref_B->BusInput3.bdcCbv.rPos_max;
  }

  /* Sum: '<S388>/Sum2' incorporates:
   *  Saturate: '<S388>/Saturation'
   *  Sum: '<S752>/Sum2'
   *  Switch: '<S752>/Switch2'
   *  Switch: '<S755>/Switch2'
   */
  rtb_LogicalOperator1_js_tmp = Gen2_ref_B->BusInput3.bdcTv.rPos_min +
    rtb_PactOut;

  /* Logic: '<S388>/Logical Operator1' incorporates:
   *  Delay: '<Root>/Delay4'
   *  Logic: '<S388>/Logical Operator2'
   *  Product: '<S388>/Divide'
   *  RelationalOperator: '<S388>/Relational Operator2'
   *  RelationalOperator: '<S388>/Relational Operator3'
   *  Saturate: '<S388>/Saturation1'
   *  Sum: '<S388>/Sum2'
   */
  rtb_LogicalOperator1_j = ((Gen2_ref_DWork->Delay4_DSTATE /
    rtb_deltafalllimit_ca >= rtb_Switch2_l) && ((rtb_Switch_on <=
    rtb_LogicalOperator1_js_tmp) || rtb_LogicalOperator5_mv));

  /* Switch: '<S390>/Switch2' incorporates:
   *  RelationalOperator: '<S390>/LowerRelop1'
   */
  if (!(rtb_Switch_jz > rtb_mbar2pa_g)) {
    /* Switch: '<S388>/Switch1' incorporates:
     *  Constant: '<S388>/Constant2'
     *  Constant: '<S388>/Constant3'
     */
    if (rtb_LogicalOperator1_j) {
      rtb_Switch_on = 0.0;
    } else {
      rtb_Switch_on = -1.0E+6;
    }

    /* End of Switch: '<S388>/Switch1' */

    /* Switch: '<S390>/Switch' incorporates:
     *  RelationalOperator: '<S390>/UpperRelop'
     */
    if (rtb_Switch_jz < rtb_Switch_on) {
      rtb_mbar2pa_g = rtb_Switch_on;
    } else {
      rtb_mbar2pa_g = rtb_Switch_jz;
    }

    /* End of Switch: '<S390>/Switch' */
  }

  /* End of Switch: '<S390>/Switch2' */

  /* Outputs for Atomic SubSystem: '<S6>/TOF1' */
  /* RelationalOperator: '<S6>/Relational Operator' incorporates:
   *  DataTypeConversion: '<S4>/Data Type Conversion30'
   */
  Gen2_ref_TOF((Gen2_ref_B->BusInput.rKnock_level >
                Gen2_ref_B->BusInput3.GQC.rThreshold_knock),
               Gen2_ref_B->BusInput3.GQC.rTOF_KnockMisfDet, &Gen2_ref_B->TOF1,
               &Gen2_ref_DWork->TOF1, inst);

  /* End of Outputs for SubSystem: '<S6>/TOF1' */

  /* Switch: '<S6>/Switch2' */
  rtb_Switch2_jv = (Gen2_ref_B->BusInput3.GQC.bActKnockDetGQC &&
                    Gen2_ref_B->TOF1.LogicalOperator1);

  /* Logic: '<S343>/Logical Operator2' */
  rtb_LogicalOperator2_e = !rtb_Switch2_jv;

  /* Outputs for Atomic SubSystem: '<S6>/TOF2' */
  /* RelationalOperator: '<S6>/Relational Operator1' incorporates:
   *  DataTypeConversion: '<S4>/Data Type Conversion33'
   */
  Gen2_ref_TOF((Gen2_ref_B->BusInput.rMisfire_level >
                Gen2_ref_B->BusInput3.GQC.rThreshold_misfire),
               Gen2_ref_B->BusInput3.GQC.rTOF_KnockMisfDet, &Gen2_ref_B->TOF2,
               &Gen2_ref_DWork->TOF2, inst);

  /* End of Outputs for SubSystem: '<S6>/TOF2' */

  /* Switch: '<S6>/Switch4' */
  rtb_Switch4_mu = (Gen2_ref_B->BusInput3.GQC.bActKnockDetGQC &&
                    Gen2_ref_B->TOF2.LogicalOperator1);

  /* Logic: '<S343>/Logical Operator4' */
  rtb_LogicalOperator5_mv = !rtb_Switch4_mu;

  /* Switch: '<S343>/Switch3' incorporates:
   *  UnitDelay: '<S343>/Unit Delay1'
   */
  if (rtb_LogicalOperator5_mv) {
    /* Switch: '<S343>/Switch2' incorporates:
     *  UnitDelay: '<S343>/Unit Delay1'
     */
    if (rtb_LogicalOperator2_e) {
      rtb_Switch_on = rtb_mbar2pa_g;
    } else {
      rtb_Switch_on = Gen2_ref_DWork->UnitDelay1_DSTATE;
    }

    /* End of Switch: '<S343>/Switch2' */
  } else {
    rtb_Switch_on = Gen2_ref_DWork->UnitDelay1_DSTATE;
  }

  /* End of Switch: '<S343>/Switch3' */

  /* Switch: '<S343>/Switch' */
  if (!rtb_LogicalOperator2_e) {
    /* Saturate: '<S343>/Saturation1' */
    if (rtb_mbar2pa_g < 0.0) {
      rtb_mbar2pa_g = 0.0;
    }

    /* End of Saturate: '<S343>/Saturation1' */
  }

  /* End of Switch: '<S343>/Switch' */

  /* Switch: '<S343>/Switch1' incorporates:
   *  Saturate: '<S343>/Saturation2'
   */
  if (rtb_LogicalOperator5_mv) {
    rtb_Switch_jz = rtb_mbar2pa_g;
  } else if (rtb_mbar2pa_g > 0.0) {
    /* Saturate: '<S343>/Saturation2' */
    rtb_Switch_jz = 0.0;
  } else {
    /* Saturate: '<S343>/Saturation2' */
    rtb_Switch_jz = rtb_mbar2pa_g;
  }

  /* End of Switch: '<S343>/Switch1' */

  /* DataTypeConversion: '<S343>/Data Type Conversion2' incorporates:
   *  UnitDelay: '<S343>/Unit Delay'
   */
  rtb_mbar2pa_g = Gen2_ref_DWork->UnitDelay_DSTATE_mg;

  /* Saturate: '<S343>/Saturation' */
  if (rtb_mbar2pa_g > 0.01) {
    rtb_mbar2pa_g = 0.01;
  } else if (rtb_mbar2pa_g < -0.01) {
    rtb_mbar2pa_g = -0.01;
  }

  /* End of Saturate: '<S343>/Saturation' */

  /* Product: '<S343>/Product1' incorporates:
   *  DataTypeConversion: '<S343>/Data Type Conversion1'
   *  Gain: '<S343>/Gain2'
   *  Logic: '<S343>/Logical Operator1'
   *  Logic: '<S343>/Logical Operator3'
   *  Logic: '<S388>/Logical Operator3'
   */
  rtb_Product1 = -(real_T)((!rtb_bActGasQualImprov) || (rtb_LogicalOperator1_j ||
    rtb_LogicalOperator2_p1)) * rtb_mbar2pa_g *
    Gen2_ref_B->BusInput3.PowCtrlGQCp2s.rFactAW_aux;

  /* Product: '<S343>/Product2' */
  rtb_Pa2bar_o = rtb_PactOut_o / rtb_Product1_aq;

  /* S-Function (sfix_look1_dyn): '<S343>/Lookup Table Dynamic' */
  /* Dynamic Look-Up Table Block: '<S343>/Lookup Table Dynamic'
   * Input0  Data Type:  Floating Point real_T
   * Input1  Data Type:  Floating Point real_T
   * Input2  Data Type:  Floating Point real_T
   * Output0 Data Type:  Floating Point real_T
   * Lookup Method: Linear_Endpoint
   *
   */
  LookUp_real_T_real_T( &(rtb_mbar2pa_g),
                       &Gen2_ref_B->BusInput3.PowCtrlGQCp2s.rPrP2sOffs_max_y[0],
                       rtb_Pa2bar_o,
                       &Gen2_ref_B->BusInput3.PowCtrlGQCp2s.rPrP2sOffs_max_x[0],
                       5U, inst);

  /* Gain: '<S343>/mbar2bar' */
  rtb_rKK2_k = 0.001 * rtb_mbar2pa_g;

  /* Outputs for Atomic SubSystem: '<S343>/PID_Power' */
  /* Product: '<S389>/Divide1' */
  FILT_IN = Gen2_ref_B->BusInput3.PowCtrlGQCp2s.rKp * rtb_Switch_on;

  /* BusCreator: '<Root>/Bus Creator' incorporates:
   *  DataTypeConversion: '<S389>/Data Type Conversion1'
   *  Outport: '<Root>/dbg'
   */
  Gen2_ref_Y->dbg.HLC.dbgHLCPowCtrlGQC.up = (real32_T)FILT_IN;

  /* Product: '<S389>/Divide2' */
  r = rtb_Switch_jz * Gen2_ref_B->BusInput3.PowCtrlGQCp2s.rKd;

  /* DiscreteIntegrator: '<S389>/Discrete-Time Integrator1' */
  if (rtb_LogicalOperator_in || (Gen2_ref_DWork->DiscreteTimeIntegrator1_Prev_ko
       != 0)) {
    Gen2_ref_DWork->DiscreteTimeIntegrator1_DSTAT_m = 0.0;
  }

  /* Product: '<S389>/Divide3' incorporates:
   *  DiscreteIntegrator: '<S389>/Discrete-Time Integrator1'
   *  Sum: '<S389>/Sum1'
   */
  rtb_Divide3_d = (r - Gen2_ref_DWork->DiscreteTimeIntegrator1_DSTAT_m) *
    Gen2_ref_B->BusInput3.PowCtrlGQCp2s.rN;

  /* Delay: '<S389>/Delay2' */
  r = Gen2_ref_DWork->Delay2_DSTATE_h;

  /* MATLAB Function: '<S389>/MATLAB Function' incorporates:
   *  Constant: '<S343>/Constant'
   *  Sum: '<S389>/Sum6'
   */
  Gen2_ref_MATLABFunction_g(rtb_LogicalOperator_in, 0.0, rtb_LogicalOperator1_e,
    (r - FILT_IN) - rtb_Divide3_d, &Gen2_ref_B->sf_MATLABFunction_a,
    &Gen2_ref_DWork->sf_MATLABFunction_a, inst);

  /* DiscreteIntegrator: '<S389>/Discrete-Time Integrator' */
  if (Gen2_ref_DWork->DiscreteTimeIntegrator_IC_LOA_c != 0) {
    Gen2_ref_DWork->DiscreteTimeIntegrator_DSTAT_hn =
      Gen2_ref_B->sf_MATLABFunction_a.Y0Out;
  }

  if (Gen2_ref_B->sf_MATLABFunction_a.ireset ||
      (Gen2_ref_DWork->DiscreteTimeIntegrator_PrevRe_b != 0)) {
    Gen2_ref_DWork->DiscreteTimeIntegrator_DSTAT_hn =
      Gen2_ref_B->sf_MATLABFunction_a.Y0Out;
  }

  /* Sum: '<S389>/Sum3' incorporates:
   *  DiscreteIntegrator: '<S389>/Discrete-Time Integrator'
   *  Sum: '<S389>/Sum'
   */
  FILT_IN = (FILT_IN + Gen2_ref_DWork->DiscreteTimeIntegrator_DSTAT_hn) +
    rtb_Divide3_d;

  /* Product: '<S394>/delta rise limit' incorporates:
   *  SampleTimeMath: '<S394>/sample time'
   *
   * About '<S394>/sample time':
   *  y = K where K = ( w * Ts )
   */
  r = Gen2_ref_B->BusInput3.PowCtrlGQCp2s.rLam_Sr_Pos * 0.01;

  /* Delay: '<S394>/Delay' incorporates:
   *  Constant: '<S343>/Constant1'
   *  Delay: '<S404>/Delay'
   */
  Gen2_ref_DWork->icLoad_ht = ((((Gen2_ref_PrevZCSigState->Delay_Reset_ZCE_e ==
    1) != (int32_T)rtb_LogicalOperator_in) &&
    (Gen2_ref_PrevZCSigState->Delay_Reset_ZCE_e != 3)) || rtb_LogicalOperator_in
    || Gen2_ref_DWork->icLoad_ht);
  Gen2_ref_PrevZCSigState->Delay_Reset_ZCE_e = rtb_LogicalOperator_in;
  if (Gen2_ref_DWork->icLoad_ht) {
    Gen2_ref_DWork->Delay_DSTATE_fo = 0.0;
  }

  /* Switch: '<S394>/etaVolConst' incorporates:
   *  Constant: '<S343>/Constant1'
   */
  if (rtb_LogicalOperator_in) {
    rtb_Abs = 0.0;
  } else {
    rtb_Abs = FILT_IN;
  }

  /* End of Switch: '<S394>/etaVolConst' */

  /* Sum: '<S394>/Difference Inputs1' incorporates:
   *  Delay: '<S394>/Delay'
   */
  rtb_Divide2_a = rtb_Abs - Gen2_ref_DWork->Delay_DSTATE_fo;

  /* Switch: '<S395>/Switch2' incorporates:
   *  RelationalOperator: '<S395>/LowerRelop1'
   */
  if (!(rtb_Divide2_a > r)) {
    /* Product: '<S394>/delta fall limit' incorporates:
     *  SampleTimeMath: '<S394>/sample time'
     *
     * About '<S394>/sample time':
     *  y = K where K = ( w * Ts )
     */
    rtb_Divide_kp = Gen2_ref_B->BusInput3.PowCtrlGQCp2s.rLam_Sr_Neg * 0.01;

    /* Switch: '<S395>/Switch' incorporates:
     *  RelationalOperator: '<S395>/UpperRelop'
     */
    if (rtb_Divide2_a < rtb_Divide_kp) {
      r = rtb_Divide_kp;
    } else {
      r = rtb_Divide2_a;
    }

    /* End of Switch: '<S395>/Switch' */
  }

  /* End of Switch: '<S395>/Switch2' */

  /* Sum: '<S394>/Difference Inputs2' incorporates:
   *  Delay: '<S394>/Delay'
   */
  rtb_Divide2_a = r + Gen2_ref_DWork->Delay_DSTATE_fo;

  /* Switch: '<S393>/Switch2' incorporates:
   *  RelationalOperator: '<S393>/LowerRelop1'
   */
  if (!(rtb_Divide2_a > rtb_rKK2_k)) {
    /* Gain: '<S343>/Pa2bar1' */
    rtb_rKK2_k = -rtb_rKK2_k;

    /* Switch: '<S393>/Switch' incorporates:
     *  RelationalOperator: '<S393>/UpperRelop'
     */
    if (!(rtb_Divide2_a < rtb_rKK2_k)) {
      rtb_rKK2_k = rtb_Divide2_a;
    }

    /* End of Switch: '<S393>/Switch' */
  }

  /* End of Switch: '<S393>/Switch2' */

  /* Sum: '<S389>/Sum2' */
  r = rtb_rKK2_k - FILT_IN;

  /* Product: '<S389>/Divide4' */
  r *= Gen2_ref_B->BusInput3.PowCtrlGQCp2s.rKaw;

  /* MATLAB Function: '<S389>/MATLAB Function1' */
  Gen2_ref_MATLABFunction1(rtb_rKK2_k, rtb_LogicalOperator1_e,
    &Gen2_ref_B->sf_MATLABFunction1_ep, &Gen2_ref_DWork->sf_MATLABFunction1_ep, inst);

  /* BusCreator: '<S389>/Bus Creator1' incorporates:
   *  DataTypeConversion: '<S389>/Data Type Conversion2'
   *  DiscreteIntegrator: '<S389>/Discrete-Time Integrator'
   */
  rtb_BusCreator1_h_ui = (real32_T)
    Gen2_ref_DWork->DiscreteTimeIntegrator_DSTAT_hn;

  /* BusCreator: '<Root>/Bus Creator' incorporates:
   *  BusCreator: '<S389>/Bus Creator1'
   *  DataTypeConversion: '<S389>/Data Type Conversion4'
   *  DataTypeConversion: '<S389>/Data Type Conversion7'
   *  Outport: '<Root>/dbg'
   */
  Gen2_ref_Y->dbg.HLC.dbgHLCPowCtrlGQC.aw = (real32_T)r;
  Gen2_ref_Y->dbg.HLC.dbgHLCPowCtrlGQC.u_unsat = (real32_T)FILT_IN;

  /* Product: '<S389>/Divide' */
  FILT_IN = rtb_Switch_jz * Gen2_ref_B->BusInput3.PowCtrlGQCp2s.rKi;

  /* Update for DiscreteIntegrator: '<S389>/Discrete-Time Integrator1' */
  Gen2_ref_DWork->DiscreteTimeIntegrator1_DSTAT_m += 0.01 * rtb_Divide3_d;
  Gen2_ref_DWork->DiscreteTimeIntegrator1_Prev_ko = (int8_T)
    rtb_LogicalOperator_in;

  /* Update for Delay: '<S389>/Delay2' */
  Gen2_ref_DWork->Delay2_DSTATE_h = Gen2_ref_B->sf_MATLABFunction1_ep.LamOut;

  /* Update for DiscreteIntegrator: '<S389>/Discrete-Time Integrator' incorporates:
   *  Sum: '<S389>/Sum4'
   *  Sum: '<S389>/Sum5'
   */
  Gen2_ref_DWork->DiscreteTimeIntegrator_IC_LOA_c = 0U;
  Gen2_ref_DWork->DiscreteTimeIntegrator_DSTAT_hn += ((rtb_Product1 + r) +
    FILT_IN) * 0.01;
  Gen2_ref_DWork->DiscreteTimeIntegrator_PrevRe_b = (int8_T)
    Gen2_ref_B->sf_MATLABFunction_a.ireset;

  /* Update for Delay: '<S394>/Delay' */
  Gen2_ref_DWork->icLoad_ht = false;
  Gen2_ref_DWork->Delay_DSTATE_fo = rtb_Divide2_a;

  /* End of Outputs for SubSystem: '<S343>/PID_Power' */

  /* Sum: '<S345>/Sum1' incorporates:
   *  Constant: '<S345>/Constant1'
   *  DiscreteIntegrator: '<S345>/Discrete-Time Integrator'
   *  Gain: '<S343>/2Pa'
   *  Product: '<S345>/Product'
   *  Product: '<S345>/Product1'
   *  Sum: '<S345>/Sum'
   *  Sum: '<S7>/Sum'
   */
  rtb_Pa2bar_o = (100000.0 * Gen2_ref_B->sf_MATLABFunction1_ep.LamOut +
                  rtb_Pa2bar_k) * Gen2_ref_DWork->DiscreteTimeIntegrator_DSTATE
    + (1.0 - Gen2_ref_DWork->DiscreteTimeIntegrator_DSTATE) *
    Gen2_ref_B->p2sfilt.Switch;

  /* Product: '<S795>/delta rise limit' */
  rtb_mbar2pa_g = rtb_Divide_mr_tmp_0;

  /* DiscreteIntegrator: '<S760>/Discrete-Time Integrator' */
  if (rtb_bResetHlci || (Gen2_ref_DWork->DiscreteTimeIntegrator_PrevRe_i != 0))
  {
    Gen2_ref_DWork->DiscreteTimeIntegrator_DSTATE_h = 1.0;
  }

  if (Gen2_ref_DWork->DiscreteTimeIntegrator_DSTATE_h >= 1.0) {
    Gen2_ref_DWork->DiscreteTimeIntegrator_DSTATE_h = 1.0;
  } else if (Gen2_ref_DWork->DiscreteTimeIntegrator_DSTATE_h <= 0.0) {
    Gen2_ref_DWork->DiscreteTimeIntegrator_DSTATE_h = 0.0;
  }

  /* Logic: '<S760>/Logical Operator' incorporates:
   *  Constant: '<S760>/Constant2'
   *  DiscreteIntegrator: '<S760>/Discrete-Time Integrator'
   *  RelationalOperator: '<S760>/Relational Operator'
   */
  rtb_LogicalOperator1_j = ((0.99 <=
    Gen2_ref_DWork->DiscreteTimeIntegrator_DSTATE_h) || rtb_bResetHlci);

  /* Delay: '<S795>/Delay' */
  Gen2_ref_DWork->icLoad_h = ((((Gen2_ref_PrevZCSigState->Delay_Reset_ZCE_m == 1)
    != (int32_T)rtb_LogicalOperator1_j) &&
    (Gen2_ref_PrevZCSigState->Delay_Reset_ZCE_m != 3)) || rtb_LogicalOperator1_j
    || Gen2_ref_DWork->icLoad_h);
  Gen2_ref_PrevZCSigState->Delay_Reset_ZCE_m = rtb_LogicalOperator1_j;
  if (Gen2_ref_DWork->icLoad_h) {
    Gen2_ref_DWork->Delay_DSTATE_b = rtb_bar2Pa6;
  }

  /* Sum: '<S795>/Difference Inputs1' incorporates:
   *  Delay: '<S795>/Delay'
   *  Switch: '<S795>/etaVolConst'
   */
  rtb_Switch_jz = rtb_bar2Pa6 - Gen2_ref_DWork->Delay_DSTATE_b;

  /* Switch: '<S798>/Switch2' incorporates:
   *  RelationalOperator: '<S798>/LowerRelop1'
   */
  if (!(rtb_Switch_jz > rtb_mbar2pa_g)) {
    /* Product: '<S795>/delta fall limit' incorporates:
     *  Gain: '<S760>/Gain15'
     *  SampleTimeMath: '<S795>/sample time'
     *
     * About '<S795>/sample time':
     *  y = K where K = ( w * Ts )
     */
    rtb_rKK2_k = -rtb_Switch_ct_tmp * 0.01;

    /* Switch: '<S798>/Switch' incorporates:
     *  RelationalOperator: '<S798>/UpperRelop'
     */
    if (rtb_Switch_jz < rtb_rKK2_k) {
      rtb_mbar2pa_g = rtb_rKK2_k;
    } else {
      rtb_mbar2pa_g = rtb_Switch_jz;
    }

    /* End of Switch: '<S798>/Switch' */
  }

  /* End of Switch: '<S798>/Switch2' */

  /* Sum: '<S795>/Difference Inputs2' incorporates:
   *  Delay: '<S795>/Delay'
   */
  rtb_Switch_jz = rtb_mbar2pa_g + Gen2_ref_DWork->Delay_DSTATE_b;

  /* Outputs for Atomic SubSystem: '<S760>/p2sfilt' */
  Gen2_ref_N_TC_HP_filt(rtb_Switch_jz,
                        Gen2_ref_B->BusInput3.traj.rTiF_Pr_p2s_Man,
                        rtb_LogicalOperator1_j, &Gen2_ref_B->p2sfilt_l,
                        &Gen2_ref_DWork->p2sfilt_l, inst);

  /* End of Outputs for SubSystem: '<S760>/p2sfilt' */

  /* Gain: '<S432>/bar2mbar1' incorporates:
   *  Gain: '<S430>/bar2mbar1'
   */
  rtb_mbar2pa_i = 1000.0 * Gen2_ref_B->BusInput3.traj.rPr_p2s_max;
  rtb_mbar2pa_g = rtb_mbar2pa_i;

  /* Sum: '<S424>/Sum4' incorporates:
   *  Constant: '<S424>/Constant2'
   */
  rtb_Switch2_l = Gen2_ref_B->BusInput3.SpeedCtrl.rLSLff2load_lim + 1.0;

  /* Outputs for Atomic SubSystem: '<S424>/speed Filter' */
  Gen2_ref_N_TC_HP_filt(rtb_Switch_i5[0],
                        Gen2_ref_B->BusInput3.SpeedCtrl.rTiF_SpeedffRefDroop,
                        rtb_bResetHlci, &Gen2_ref_B->speedFilter,
                        &Gen2_ref_DWork->speedFilter, inst);

  /* End of Outputs for SubSystem: '<S424>/speed Filter' */

  /* Switch: '<S424>/Switch1' */
  if (Gen2_ref_B->BusInput3.SpeedCtrl.bffRefDroopMeasSpeed) {
    /* Switch: '<S424>/Switch2' */
    if (Gen2_ref_B->BusInput3.SpeedCtrl.bffRefDroopFiltMeasSpd) {
      rtb_bResetHlci_0 = Gen2_ref_B->speedFilter.Switch;
    } else {
      rtb_bResetHlci_0 = rtb_Switch_i5[0];
    }

    /* End of Switch: '<S424>/Switch2' */
  } else {
    rtb_bResetHlci_0 = Gen2_ref_B->BusInput3.eng.rN_Nom;
  }

  /* End of Switch: '<S424>/Switch1' */

  /* Sum: '<S424>/Sum2' */
  rtb_rKK2_k = rtb_Switch_i5[1] - rtb_bResetHlci_0;

  /* Outputs for Atomic SubSystem: '<S424>/Filter1' */
  Gen2_ref_Filter1(rtb_rKK2_k, Gen2_ref_B->BusInput3.SpeedCtrl.rTiF_LSLff_d,
                   rtb_bResetHlci, &Gen2_ref_B->Filter1_f,
                   &Gen2_ref_DWork->Filter1_f, inst);

  /* End of Outputs for SubSystem: '<S424>/Filter1' */

  /* Product: '<S424>/Divide2' */
  rtb_Divide2_a = Gen2_ref_B->Filter1_f.Switch1 *
    Gen2_ref_B->BusInput3.SpeedCtrl.rLSLff2load_d;

  /* Saturate: '<S424>/Saturation' */
  if (Gen2_ref_B->BusInput3.eng.rN_Nom <= 1.0) {
    rtb_bResetHlci_0 = 1.0;
  } else {
    rtb_bResetHlci_0 = Gen2_ref_B->BusInput3.eng.rN_Nom;
  }

  /* End of Saturate: '<S424>/Saturation' */

  /* Product: '<S424>/Divide' */
  rtb_Divide_kp = rtb_rKK2_k / rtb_bResetHlci_0 *
    Gen2_ref_B->BusInput3.SpeedCtrl.rLSLff2load;

  /* Product: '<S424>/Divide1' incorporates:
   *  Constant: '<S424>/Constant'
   *  Sum: '<S424>/Sum3'
   */
  rtb_rKK2_k = ((rtb_Divide2_a + rtb_Divide_kp) + 1.0) *
    Gen2_ref_B->BusInput3.SpeedCtrl.rff2load_Ext;

  /* Switch: '<S479>/Switch2' incorporates:
   *  RelationalOperator: '<S479>/LowerRelop1'
   */
  if (rtb_rKK2_k > rtb_Switch2_l) {
    rtb_Sum1_jz = rtb_Switch2_l;
  } else {
    /* Sum: '<S424>/Sum1' incorporates:
     *  Constant: '<S424>/Constant1'
     */
    rtb_Sum1_jz = 1.0 - Gen2_ref_B->BusInput3.SpeedCtrl.rLSLff2load_lim;

    /* Switch: '<S479>/Switch' incorporates:
     *  Constant: '<S424>/Constant1'
     *  RelationalOperator: '<S479>/UpperRelop'
     *  Sum: '<S424>/Sum1'
     */
    if (!(rtb_rKK2_k < 1.0 - Gen2_ref_B->BusInput3.SpeedCtrl.rLSLff2load_lim)) {
      rtb_Sum1_jz = rtb_rKK2_k;
    }

    /* End of Switch: '<S479>/Switch' */
  }

  /* End of Switch: '<S479>/Switch2' */

  /* Saturate: '<S761>/Saturation2' */
  if (rtb_Switch_i5[2] > 1.0) {
    rtb_rKK2_k = 1.0;
  } else if (rtb_Switch_i5[2] < 0.1) {
    rtb_rKK2_k = 0.1;
  } else {
    rtb_rKK2_k = rtb_Switch_i5[2];
  }

  /* End of Saturate: '<S761>/Saturation2' */

  /* Outputs for Atomic SubSystem: '<S761>/Filter1' */
  /* UnitDelay: '<S761>/Unit Delay2' */
  Gen2_ref_Filter3(Gen2_ref_DWork->UnitDelay2_DSTATE,
                   Gen2_ref_B->BusInput3.LoadEst.rTiFCorrUnom,
                   Gen2_ref_ConstB.Constant1_g, rtb_bResetHlci,
                   &Gen2_ref_B->Filter1_p, &Gen2_ref_DWork->Filter1_p, inst);

  /* End of Outputs for SubSystem: '<S761>/Filter1' */

  /* Sum: '<S761>/Sum1' */
  rtb_Switch_iy = rtb_rKK2_k + Gen2_ref_B->Filter1_p.Switch;

  /* Math: '<S761>/Math Function1' */
  if ((rtb_Switch_iy < 0.0) && (Gen2_ref_B->BusInput3.LoadEst.rNu > floor
       (Gen2_ref_B->BusInput3.LoadEst.rNu))) {
    rtb_Switch_iy = -rt_powd_snf(-rtb_Switch_iy,
      Gen2_ref_B->BusInput3.LoadEst.rNu, inst);
  } else {
    rtb_Switch_iy = rt_powd_snf(rtb_Switch_iy, Gen2_ref_B->BusInput3.LoadEst.rNu, inst);
  }

  /* End of Math: '<S761>/Math Function1' */

  /* Abs: '<S799>/Abs' */
  rtb_Switch2_l = fabs(rtb_Switch_iy);

  /* Switch: '<S799>/Switch' incorporates:
   *  Constant: '<S799>/Constant2'
   *  RelationalOperator: '<S799>/Relational Operator'
   */
  if (2.2204460492503131E-16 >= rtb_Switch2_l) {
    rtb_Switch_iy = 2.2204460492503131E-16;
  }

  /* End of Switch: '<S799>/Switch' */

  /* Switch: '<S761>/Switch2' incorporates:
   *  Constant: '<S761>/Constant2'
   *  Product: '<S761>/Divide'
   *  Product: '<S761>/Divide1'
   *  Product: '<S761>/Divide2'
   *  Sum: '<S761>/Sum2'
   *  Sum: '<S761>/Sum3'
   */
  if (Gen2_ref_B->BusInput3.SpeedCtrl.bAddLSLfac) {
    rtb_Switch2_gs = (rtb_Sum1_jz - 1.0) * rtb_Product1_aq + rtb_Switch_i5[3] /
      rtb_Switch_iy;
  } else {
    rtb_Switch2_gs = rtb_Switch_i5[3] / rtb_Switch_iy * rtb_Sum1_jz;
  }

  /* Outputs for Atomic SubSystem: '<S761>/Filter' */
  Gen2_ref_Pd_filt(rtb_Switch2_gs, Gen2_ref_B->BusInput3.LoadEst.rTiF_PowEst,
                   rtb_Switch_i5[3], rtb_bResetHlci, &Gen2_ref_B->Filter_kj,
                   &Gen2_ref_DWork->Filter_kj, inst);

  /* End of Outputs for SubSystem: '<S761>/Filter' */

  /* Switch: '<S761>/Switch' */
  if (Gen2_ref_B->BusInput3.LoadEst.bFilterOFF) {
    rtb_Switch_bs = rtb_Switch2_gs;
  } else {
    rtb_Switch_bs = Gen2_ref_B->Filter_kj.Switch;
  }

  /* End of Switch: '<S761>/Switch' */

  /* Gain: '<S758>/W2kW' */
  rtb_W2kW_o = 0.001 * rtb_Switch_bs;

  /* Switch: '<S792>/Switch2' incorporates:
   *  RelationalOperator: '<S792>/LowerRelop1'
   */
  if (rtb_W2kW_o > Gen2_ref_B->BusInput3.eng.rP_Nom) {
    rtb_Divide6_n = Gen2_ref_B->BusInput3.eng.rP_Nom;
  } else {
    /* Product: '<S789>/Divide6' */
    rtb_Divide6_n = Gen2_ref_B->BusInput3.eng.rP_Nom *
      Gen2_ref_B->BusInput3.leanox.rP_P2sRedIP_SP_Norm;

    /* Switch: '<S792>/Switch' incorporates:
     *  RelationalOperator: '<S792>/UpperRelop'
     */
    if (!(rtb_W2kW_o < rtb_Divide6_n)) {
      rtb_Divide6_n = rtb_W2kW_o;
    }

    /* End of Switch: '<S792>/Switch' */
  }

  /* End of Switch: '<S792>/Switch2' */

  /* MATLAB Function: '<S789>/2-point interpolation, with extrapolation' */
  upointinterpolationwithextrapol(rtb_Divide6_n,
    Gen2_ref_B->BusInput3.leanox.Comp_IgnP_x,
    Gen2_ref_B->BusInput3.leanox.Comp_IgnP_y,
    &Gen2_ref_B->sf_2pointinterpolationwithext_a, inst);

  /* Switch: '<S789>/Switch1' incorporates:
   *  Constant: '<S789>/Pel_a (kW)1'
   *  DataTypeConversion: '<S4>/Data Type Conversion22'
   *  Product: '<S789>/Divide5'
   *  Sum: '<S789>/Add12'
   */
  if (Gen2_ref_B->BusInput3.leanox.bZZPKorr) {
    rtb_Switch2_l = (Gen2_ref_B->BusInput.rCA_Ign_OP_Power -
                     Gen2_ref_B->N_TC_HP_filt.Switch) *
      Gen2_ref_B->sf_2pointinterpolationwithext_a.y;
  } else {
    rtb_Switch2_l = 0.0;
  }

  /* End of Switch: '<S789>/Switch1' */

  /* Switch: '<S793>/Switch2' incorporates:
   *  RelationalOperator: '<S793>/LowerRelop1'
   */
  if (rtb_W2kW_o > Gen2_ref_B->BusInput3.eng.rP_Nom) {
    rtb_Divide6_n = Gen2_ref_B->BusInput3.eng.rP_Nom;
  } else {
    /* Product: '<S789>/Divide1' */
    rtb_Divide6_n = Gen2_ref_B->BusInput3.eng.rP_Nom *
      Gen2_ref_B->BusInput3.leanox.rP2s_Comp_Act_SP;

    /* Switch: '<S793>/Switch' incorporates:
     *  RelationalOperator: '<S793>/UpperRelop'
     */
    if (!(rtb_W2kW_o < rtb_Divide6_n)) {
      rtb_Divide6_n = rtb_W2kW_o;
    }

    /* End of Switch: '<S793>/Switch' */
  }

  /* End of Switch: '<S793>/Switch2' */

  /* MATLAB Function: '<S789>/2-point interpolation, with extrapolation1' */
  upointinterpolationwithextrapol(rtb_Divide6_n,
    Gen2_ref_B->BusInput3.leanox.Comp_ChTmp_x,
    Gen2_ref_B->BusInput3.leanox.Comp_ChTmp_y,
    &Gen2_ref_B->sf_2pointinterpolationwithex_je, inst);

  /* Switch: '<S789>/Switch2' incorporates:
   *  Constant: '<S789>/Pel_a (kW)2'
   *  Product: '<S789>/Divide9'
   *  Sum: '<S789>/Add13'
   */
  if (Gen2_ref_B->BusInput3.leanox.bt2Korr) {
    rtb_bResetHlci_0 = (Gen2_ref_B->T2s_filt.Switch -
                        Gen2_ref_B->BusInput3.leanox.rT_2) *
      Gen2_ref_B->sf_2pointinterpolationwithex_je.y;
  } else {
    rtb_bResetHlci_0 = 0.0;
  }

  /* End of Switch: '<S789>/Switch2' */

  /* Switch: '<S789>/Switch3' incorporates:
   *  Constant: '<S789>/Pel_a (kW)3'
   */
  if (Gen2_ref_B->BusInput3.leanox.bHum_Act) {
    delta_y = Gen2_ref_B->BusInput3.leanox.rP2s_Comp_HumOffset;
  } else {
    delta_y = 0.0;
  }

  /* End of Switch: '<S789>/Switch3' */

  /* Sum: '<S775>/Add11' */
  rtb_Divide6_n = (rtb_Switch2_l + rtb_bResetHlci_0) + delta_y;

  /* Switch: '<S758>/Switch1' incorporates:
   *  Product: '<S758>/Divide6'
   *  Sum: '<S758>/Add4'
   */
  if (Gen2_ref_B->BusInput.tLEANOXin.bZylAusfall) {
    /* Switch: '<S771>/Switch' incorporates:
     *  Abs: '<S771>/Abs'
     *  Constant: '<S771>/Constant2'
     *  RelationalOperator: '<S771>/Relational Operator'
     */
    if (1.0 >= fabs(Gen2_ref_B->BusInput3.eng.rNum_Cyl_Eng)) {
      rtb_bResetHlci_0 = 1.0;
    } else {
      rtb_bResetHlci_0 = Gen2_ref_B->BusInput3.eng.rNum_Cyl_Eng;
    }

    /* End of Switch: '<S771>/Switch' */
    rtb_Switch1_k = rtb_W2kW_o / rtb_bResetHlci_0 + rtb_W2kW_o;
  } else {
    rtb_Switch1_k = rtb_W2kW_o;
  }

  /* End of Switch: '<S758>/Switch1' */

  /* Switch: '<S432>/Switch' */
  if (Gen2_ref_B->BusInput3.SpeedCtrl.bRefSpeedLEANOX) {
    rtb_Switch2_n5 = rtb_Switch_i5[1];
  } else {
    rtb_Switch2_n5 = Gen2_ref_B->BusInput3.eng.rN_Nom;
  }

  /* End of Switch: '<S432>/Switch' */

  /* Switch: '<S762>/Switch' incorporates:
   *  Abs: '<S762>/Abs'
   *  Constant: '<S762>/Constant2'
   *  RelationalOperator: '<S762>/Relational Operator'
   */
  if (1.0 >= fabs(rtb_Switch2_n5)) {
    rtb_Switch2_n5 = 1.0;
  }

  /* End of Switch: '<S762>/Switch' */

  /* Switch: '<S758>/Switch4' */
  if (Gen2_ref_B->BusInput3.leanox.bLp_c_Ena) {
    rtb_bResetHlci_0 = Gen2_ref_B->BusInput3.leanox.rP_c;
  } else {
    rtb_bResetHlci_0 = Gen2_ref_B->BusInput3.leanox.rP_1;
  }

  /* End of Switch: '<S758>/Switch4' */

  /* Switch: '<S758>/Switch2' incorporates:
   *  Logic: '<S758>/Logical Operator1'
   *  Product: '<S758>/Divide4'
   *  RelationalOperator: '<S758>/Relational Operator1'
   *  RelationalOperator: '<S758>/Relational Operator3'
   *  Sum: '<S758>/Add5'
   *  Switch: '<S758>/Switch5'
   */
  if (rtb_Switch1_k < rtb_bResetHlci_0) {
    /* Switch: '<S758>/Switch_b_c' incorporates:
     *  Logic: '<S758>/Logical Operator'
     *  RelationalOperator: '<S758>/Relational Operator2'
     */
    if (Gen2_ref_B->BusInput3.leanox.bLp_c_Ena && (rtb_Switch1_k <
         Gen2_ref_B->BusInput3.leanox.rP_c)) {
      /* SignalConversion generated from: '<S758>/Lookup Table Dynamic1' */
      rtb_TmpSignalConversionAtLoo_ht[0] =
        Gen2_ref_B->BusInput3.leanox.rPr_mbar_0;

      /* Switch: '<S772>/Switch' incorporates:
       *  Abs: '<S772>/Abs'
       *  Constant: '<S772>/Constant2'
       *  RelationalOperator: '<S772>/Relational Operator'
       */
      if (1.0 >= fabs(Gen2_ref_B->BusInput3.leanox.rT_c)) {
        rtb_bResetHlci_0 = 1.0;
      } else {
        rtb_bResetHlci_0 = Gen2_ref_B->BusInput3.leanox.rT_c;
      }

      /* End of Switch: '<S772>/Switch' */

      /* SignalConversion generated from: '<S758>/Lookup Table Dynamic1' incorporates:
       *  Product: '<S758>/Divide5'
       */
      rtb_TmpSignalConversionAtLoo_ht[1] =
        Gen2_ref_B->BusInput3.leanox.rPr_mbar_c *
        Gen2_ref_B->BusInput3.leanox.rN_c / rtb_bResetHlci_0 *
        Gen2_ref_B->T2s_filt.Switch / rtb_Switch2_n5;

      /* SignalConversion generated from: '<S758>/Lookup Table Dynamic1' incorporates:
       *  Constant: '<S758>/Pel_a (kW)1'
       */
      rtb_TmpSignalConversionAtLook_d[0] = 0.0;
      rtb_TmpSignalConversionAtLook_d[1] = Gen2_ref_B->BusInput3.leanox.rP_c;

      /* S-Function (sfix_look1_dyn): '<S758>/Lookup Table Dynamic1' */
      /* Dynamic Look-Up Table Block: '<S758>/Lookup Table Dynamic1'
       * Input0  Data Type:  Floating Point real_T
       * Input1  Data Type:  Floating Point real_T
       * Input2  Data Type:  Floating Point real_T
       * Output0 Data Type:  Floating Point real_T
       * Lookup Method: Linear_Endpoint
       *
       */
      LookUp_real_T_real_T( &(rtb_LookupTableDynamic1_b),
                           &rtb_TmpSignalConversionAtLoo_ht[0], rtb_Switch1_k,
                           &rtb_TmpSignalConversionAtLook_d[0], 1U, inst);
      rtb_Switch2_n5 = rtb_LookupTableDynamic1_b;
    } else {
      /* SignalConversion generated from: '<S758>/Lookup Table Dynamic' */
      rtb_TmpSignalConversionAtLoo_ht[0] =
        Gen2_ref_B->BusInput3.leanox.rPr_mbar_0;

      /* Switch: '<S770>/Switch' incorporates:
       *  Abs: '<S770>/Abs'
       *  Constant: '<S770>/Constant2'
       *  RelationalOperator: '<S770>/Relational Operator'
       */
      if (1.0 >= fabs(Gen2_ref_B->BusInput3.leanox.rT_1)) {
        rtb_bResetHlci_0 = 1.0;
      } else {
        rtb_bResetHlci_0 = Gen2_ref_B->BusInput3.leanox.rT_1;
      }

      /* End of Switch: '<S770>/Switch' */

      /* SignalConversion generated from: '<S758>/Lookup Table Dynamic' incorporates:
       *  Product: '<S758>/Divide1'
       */
      rtb_TmpSignalConversionAtLoo_ht[1] =
        Gen2_ref_B->BusInput3.leanox.rPr_mbar_1 *
        Gen2_ref_B->BusInput3.leanox.rN_1 / rtb_bResetHlci_0 *
        Gen2_ref_B->T2s_filt.Switch / rtb_Switch2_n5;

      /* SignalConversion generated from: '<S758>/Lookup Table Dynamic' incorporates:
       *  Constant: '<S758>/Pel_a (kW)3'
       */
      rtb_TmpSignalConversionAtLook_d[0] = 0.0;
      rtb_TmpSignalConversionAtLook_d[1] = Gen2_ref_B->BusInput3.leanox.rP_1;

      /* S-Function (sfix_look1_dyn): '<S758>/Lookup Table Dynamic' */
      /* Dynamic Look-Up Table Block: '<S758>/Lookup Table Dynamic'
       * Input0  Data Type:  Floating Point real_T
       * Input1  Data Type:  Floating Point real_T
       * Input2  Data Type:  Floating Point real_T
       * Output0 Data Type:  Floating Point real_T
       * Lookup Method: Linear_Endpoint
       *
       */
      LookUp_real_T_real_T( &(rtb_LookupTableDynamic_m),
                           &rtb_TmpSignalConversionAtLoo_ht[0], rtb_Switch1_k,
                           &rtb_TmpSignalConversionAtLook_d[0], 1U, inst);
      rtb_Switch2_n5 = rtb_LookupTableDynamic_m;
    }

    /* End of Switch: '<S758>/Switch_b_c' */
  } else {
    if (Gen2_ref_B->BusInput3.leanox.bLp_c_Ena && (rtb_Switch1_k <
         Gen2_ref_B->BusInput3.leanox.rP_1)) {
      /* Sum: '<S758>/Add1' incorporates:
       *  Switch: '<S758>/Switch5'
       */
      rtb_Switch_jv = Gen2_ref_B->BusInput3.leanox.rP_1 -
        Gen2_ref_B->BusInput3.leanox.rP_c;

      /* Sum: '<S758>/Sum4' incorporates:
       *  Switch: '<S758>/Switch5'
       */
      rtb_Switch_fi = Gen2_ref_B->BusInput3.leanox.rP_c +
        Gen2_ref_B->BusInput3.leanox.rP_Eng_Frict;

      /* Switch: '<S765>/Switch' incorporates:
       *  Abs: '<S765>/Abs'
       *  Constant: '<S765>/Constant2'
       *  RelationalOperator: '<S765>/Relational Operator'
       *  Switch: '<S758>/Switch5'
       */
      if (1.0 >= fabs(rtb_Switch_fi)) {
        rtb_PactOut_o = 1.0;
      } else {
        rtb_PactOut_o = rtb_Switch_fi;
      }

      /* End of Switch: '<S765>/Switch' */

      /* Sum: '<S758>/Sum5' incorporates:
       *  Switch: '<S758>/Switch5'
       */
      rtb_Switch_fi = Gen2_ref_B->BusInput3.leanox.rP_1 +
        Gen2_ref_B->BusInput3.leanox.rP_Eng_Frict;

      /* Switch: '<S773>/Switch' incorporates:
       *  Abs: '<S773>/Abs'
       *  Constant: '<S773>/Constant2'
       *  RelationalOperator: '<S773>/Relational Operator'
       *  Switch: '<S758>/Switch5'
       */
      if (1.0 >= fabs(Gen2_ref_B->BusInput3.leanox.rT_1)) {
        rtb_bResetHlci_0 = 1.0;
      } else {
        rtb_bResetHlci_0 = Gen2_ref_B->BusInput3.leanox.rT_1;
      }

      /* End of Switch: '<S773>/Switch' */

      /* Switch: '<S764>/Switch' incorporates:
       *  Abs: '<S764>/Abs'
       *  Constant: '<S764>/Constant2'
       *  RelationalOperator: '<S764>/Relational Operator'
       *  Switch: '<S758>/Switch5'
       */
      if (1.0 >= fabs(rtb_Switch_fi)) {
        rtb_Switch_fi = 1.0;
      }

      /* End of Switch: '<S764>/Switch' */

      /* Product: '<S758>/rKK3' incorporates:
       *  Switch: '<S758>/Switch5'
       */
      rtb_Switch_fi = Gen2_ref_B->BusInput3.leanox.rPr_mbar_1 *
        Gen2_ref_B->BusInput3.leanox.rN_1 / rtb_bResetHlci_0 / rtb_Switch_fi;

      /* Switch: '<S766>/Switch' incorporates:
       *  Abs: '<S766>/Abs'
       *  Constant: '<S766>/Constant2'
       *  RelationalOperator: '<S766>/Relational Operator'
       *  Switch: '<S758>/Switch5'
       */
      if (1.0 >= fabs(Gen2_ref_B->BusInput3.leanox.rT_c)) {
        rtb_bResetHlci_0 = 1.0;
      } else {
        rtb_bResetHlci_0 = Gen2_ref_B->BusInput3.leanox.rT_c;
      }

      /* End of Switch: '<S766>/Switch' */

      /* Switch: '<S774>/Switch' incorporates:
       *  Abs: '<S774>/Abs'
       *  Constant: '<S774>/Constant2'
       *  RelationalOperator: '<S774>/Relational Operator'
       *  Switch: '<S758>/Switch5'
       */
      if (1.0 >= fabs(rtb_Switch_jv)) {
        rtb_Switch_jv = 1.0;
      }

      /* End of Switch: '<S774>/Switch' */

      /* Switch: '<S758>/Switch5' incorporates:
       *  Product: '<S758>/Divide10'
       *  Product: '<S758>/Divide9'
       *  Product: '<S758>/rKK4'
       *  Sum: '<S758>/Add3'
       *  Sum: '<S758>/Sum6'
       *  Sum: '<S758>/Sum7'
       */
      rtb_W2kW_o = (rtb_Switch_fi - Gen2_ref_B->BusInput3.leanox.rPr_mbar_c *
                    Gen2_ref_B->BusInput3.leanox.rN_c / rtb_bResetHlci_0 /
                    rtb_PactOut_o) / rtb_Switch_jv * (rtb_W2kW_o -
        Gen2_ref_B->BusInput3.leanox.rP_1) + rtb_Switch_fi;
    } else {
      /* Sum: '<S758>/Add10' incorporates:
       *  Switch: '<S758>/Switch5'
       */
      rtb_Switch_jv = Gen2_ref_B->BusInput3.leanox.rP_2 -
        Gen2_ref_B->BusInput3.leanox.rP_1;

      /* Sum: '<S758>/Sum' incorporates:
       *  Switch: '<S758>/Switch5'
       */
      rtb_PactOut_o = Gen2_ref_B->BusInput3.leanox.rP_1 +
        Gen2_ref_B->BusInput3.leanox.rP_Eng_Frict;

      /* Sum: '<S758>/Sum1' incorporates:
       *  Switch: '<S758>/Switch5'
       */
      rtb_Switch_fi = Gen2_ref_B->BusInput3.leanox.rP_2 +
        Gen2_ref_B->BusInput3.leanox.rP_Eng_Frict;

      /* Switch: '<S763>/Switch' incorporates:
       *  Abs: '<S763>/Abs'
       *  Constant: '<S763>/Constant2'
       *  RelationalOperator: '<S763>/Relational Operator'
       *  Switch: '<S758>/Switch5'
       */
      if (1.0 >= fabs(Gen2_ref_B->BusInput3.leanox.rT_2)) {
        rtb_bResetHlci_0 = 1.0;
      } else {
        rtb_bResetHlci_0 = Gen2_ref_B->BusInput3.leanox.rT_2;
      }

      /* End of Switch: '<S763>/Switch' */

      /* Switch: '<S768>/Switch' incorporates:
       *  Abs: '<S768>/Abs'
       *  Constant: '<S768>/Constant2'
       *  RelationalOperator: '<S768>/Relational Operator'
       *  Switch: '<S758>/Switch5'
       */
      if (1.0 >= fabs(rtb_Switch_fi)) {
        rtb_Switch_fi = 1.0;
      }

      /* End of Switch: '<S768>/Switch' */

      /* Product: '<S758>/rKK1' incorporates:
       *  Switch: '<S758>/Switch5'
       */
      rtb_Switch_fi = Gen2_ref_B->BusInput3.leanox.rPr_mbar_2 *
        Gen2_ref_B->BusInput3.leanox.rN_2 / rtb_bResetHlci_0 / rtb_Switch_fi;

      /* Switch: '<S769>/Switch' incorporates:
       *  Abs: '<S769>/Abs'
       *  Constant: '<S769>/Constant2'
       *  RelationalOperator: '<S769>/Relational Operator'
       *  Switch: '<S758>/Switch5'
       */
      if (1.0 >= fabs(rtb_PactOut_o)) {
        rtb_PactOut_o = 1.0;
      }

      /* End of Switch: '<S769>/Switch' */

      /* Switch: '<S767>/Switch' incorporates:
       *  Abs: '<S767>/Abs'
       *  Constant: '<S767>/Constant2'
       *  RelationalOperator: '<S767>/Relational Operator'
       *  Switch: '<S758>/Switch5'
       */
      if (1.0 >= fabs(rtb_Switch_jv)) {
        rtb_Switch_jv = 1.0;
      }

      /* End of Switch: '<S767>/Switch' */

      /* Switch: '<S758>/Switch5' incorporates:
       *  Product: '<S758>/Divide2'
       *  Product: '<S758>/Divide3'
       *  Product: '<S758>/rKK2'
       *  Sum: '<S758>/Add2'
       *  Sum: '<S758>/Sum2'
       *  Sum: '<S758>/Sum3'
       */
      rtb_W2kW_o = (rtb_Switch_fi - Gen2_ref_B->BusInput3.leanox.rPr_mbar_1 *
                    Gen2_ref_B->BusInput3.leanox.rN_1 /
                    Gen2_ref_B->BusInput3.leanox.rT_1 / rtb_PactOut_o) /
        rtb_Switch_jv * (rtb_W2kW_o - Gen2_ref_B->BusInput3.leanox.rP_2) +
        rtb_Switch_fi;
    }

    rtb_Switch2_n5 = rtb_W2kW_o * Gen2_ref_B->T2s_filt.Switch *
      (Gen2_ref_B->BusInput3.leanox.rP_Eng_Frict + rtb_Switch1_k) /
      rtb_Switch2_n5;
  }

  /* End of Switch: '<S758>/Switch2' */

  /* Product: '<S775>/Divide8' incorporates:
   *  DataTypeConversion: '<S775>/Data Type Conversion2'
   */
  rtb_Switch1_k = rtb_Switch2_n5 *
    Gen2_ref_B->BusInput.tLEANOXin.rLEANOX_fact_BC;

  /* Outputs for Atomic SubSystem: '<S585>/Filter1' */
  Gen2_ref_N_TC_HP_filt(rtb_Switch_i5[3],
                        Gen2_ref_B->BusInput3.SkipF.rTi_StatSkipF_FiltP,
                        rtb_bResetBdc, &Gen2_ref_B->Filter1_fg,
                        &Gen2_ref_DWork->Filter1_fg, inst);

  /* End of Outputs for SubSystem: '<S585>/Filter1' */

  /* Sum: '<S589>/Sum' */
  rtb_Switch2_l = Gen2_ref_B->BusInput3.SkipF.rNum_P0;

  /* Abs: '<S596>/Abs' */
  rtb_W2kW_o = rtb_Switch2_ba;

  /* Switch: '<S585>/Switch' */
  if (Gen2_ref_B->BusInput3.SkipF.bStatSkipF_FiltP_active) {
    rtb_bResetHlci_0 = Gen2_ref_B->Filter1_fg.Switch;
  } else {
    rtb_bResetHlci_0 = rtb_Switch_i5[3];
  }

  /* End of Switch: '<S585>/Switch' */

  /* Switch: '<S596>/Switch' incorporates:
   *  Constant: '<S596>/Constant2'
   *  RelationalOperator: '<S596>/Relational Operator'
   */
  if (2.2204460492503131E-16 >= rtb_W2kW_o) {
    rtb_Divide_mr_tmp = 2.2204460492503131E-16;
  }

  /* End of Switch: '<S596>/Switch' */

  /* Sum: '<S589>/Sum3' incorporates:
   *  Gain: '<S589>/Gain'
   *  Product: '<S589>/Divide'
   *  Product: '<S589>/Product'
   *  Sum: '<S589>/Sum2'
   */
  rtb_W2kW_o = Gen2_ref_B->BusInput3.SkipF.rNum_P0 - (0.001 * rtb_bResetHlci_0 -
    Gen2_ref_B->BusInput3.SkipF.rP_0) * (rtb_Switch2_l / rtb_Divide_mr_tmp);

  /* Switch: '<S598>/Switch2' incorporates:
   *  Constant: '<S589>/Constant1'
   *  RelationalOperator: '<S598>/LowerRelop1'
   *  RelationalOperator: '<S598>/UpperRelop'
   *  Switch: '<S598>/Switch'
   */
  if (rtb_W2kW_o > Gen2_ref_B->BusInput3.eng.rNum_Cyl_Eng) {
    rtb_W2kW_o = Gen2_ref_B->BusInput3.eng.rNum_Cyl_Eng;
  } else if (rtb_W2kW_o < 0.0) {
    /* Switch: '<S598>/Switch' incorporates:
     *  Constant: '<S589>/Constant1'
     */
    rtb_W2kW_o = 0.0;
  }

  /* End of Switch: '<S598>/Switch2' */

  /* MATLAB Function: '<S589>/MATLAB Function' */
  Gen2_ref_MATLABFunction_n(rtb_W2kW_o, Gen2_ref_B->BusInput3.SkipF.rHy_eps,
    &Gen2_ref_B->sf_MATLABFunction_n, &Gen2_ref_DWork->sf_MATLABFunction_n, inst);

  /* Gain: '<S586>/Gain1' */
  rtb_W2kW_o = rtb_Product1_aq;

  /* Switch: '<S600>/Switch' incorporates:
   *  Abs: '<S600>/Abs'
   *  Constant: '<S600>/Constant2'
   *  RelationalOperator: '<S600>/Relational Operator'
   */
  if (2.2204460492503131E-16 >= fabs(rtb_W2kW_o)) {
    rtb_W2kW_o = 2.2204460492503131E-16;
  }

  /* End of Switch: '<S600>/Switch' */

  /* Product: '<S586>/Divide' */
  rtb_Switch_jv = rtb_Switch_i5[3] / rtb_W2kW_o;

  /* S-Function (sfix_look1_dyn): '<S586>/Lookup Table Dynamic' */
  /* Dynamic Look-Up Table Block: '<S586>/Lookup Table Dynamic'
   * Input0  Data Type:  Floating Point real_T
   * Input1  Data Type:  Floating Point real_T
   * Input2  Data Type:  Floating Point real_T
   * Output0 Data Type:  Floating Point real_T
   * Lookup Method: Linear_Endpoint
   *
   */
  LookUp_real_T_real_T( &(rtb_W2kW_o), &Gen2_ref_B->BusInput3.SkipF.rLamRefSkip
                       [0], rtb_Switch_jv,
                       &Gen2_ref_B->BusInput3.SkipF.rPrefSkipNorm[0], 1U, inst);

  /* Sum: '<S586>/Sum4' incorporates:
   *  DiscreteIntegrator: '<S579>/Discrete-Time Integrator'
   */
  rtb_W2kW_o = Gen2_ref_DWork->DiscreteTimeIntegrator_DSTATE_m - rtb_W2kW_o;

  /* MinMax: '<S586>/MinMax' */
  if ((Gen2_ref_B->BusInput3.SkipF.rPrefSkipNorm[0] >=
       Gen2_ref_B->BusInput3.SkipF.rPrefSkipNorm[1]) || rtIsNaN
      (Gen2_ref_B->BusInput3.SkipF.rPrefSkipNorm[1])) {
    rtb_PactOut_o = Gen2_ref_B->BusInput3.SkipF.rPrefSkipNorm[0];
  } else {
    rtb_PactOut_o = Gen2_ref_B->BusInput3.SkipF.rPrefSkipNorm[1];
  }

  /* MATLAB Function: '<S586>/MATLAB Function' incorporates:
   *  MinMax: '<S586>/MinMax'
   */
  if (rtb_Switch_jv > rtb_PactOut_o) {
    rtb_Switch_jv = 0.0;
  } else if (rtb_Switch_jv < 0.9 * rtb_PactOut_o) {
    rtb_Switch_jv = 1.0;
  } else {
    rtb_Switch_jv = Gen2_ref_DWork->y_z;
  }

  Gen2_ref_DWork->y_z = rtb_Switch_jv;

  /* End of MATLAB Function: '<S586>/MATLAB Function' */

  /* Sum: '<S429>/Sum' incorporates:
   *  DataTypeConversion: '<S4>/Data Type Conversion34'
   *  Sum: '<S581>/Sum2'
   */
  rtb_Divide_mr_tmp = rtb_Switch_ks - Gen2_ref_B->BusInput.rN_Eng_LRskipF;

  /* Gain: '<S586>/Gain3' */
  rtb_Switch2_l = -2.0 * Gen2_ref_B->BusInput3.SkipF.rN_LevelNskip;

  /* Logic: '<S586>/Logical Operator' incorporates:
   *  Constant: '<S586>/Constant4'
   *  RelationalOperator: '<S586>/Relational Operator1'
   *  Sum: '<S429>/Sum'
   *  Sum: '<S586>/Sum6'
   */
  rtb_LogicalOperator1_j = ((1.0 - rtb_Switch_jv != 0.0) || (rtb_Divide_mr_tmp <=
    rtb_Switch2_l));

  /* DiscreteIntegrator: '<S586>/Discrete-Time Integrator' */
  if (rtb_LogicalOperator1_j || (Gen2_ref_DWork->DiscreteTimeIntegrator_PrevRe_k
       != 0)) {
    Gen2_ref_DWork->DiscreteTimeIntegrator_DSTATE_p = 0.0;
  }

  /* Product: '<S586>/Product1' incorporates:
   *  DiscreteIntegrator: '<S586>/Discrete-Time Integrator'
   *  Product: '<S586>/Product2'
   *  Sum: '<S586>/Sum9'
   */
  rtb_Switch_fi = (rtb_W2kW_o * Gen2_ref_B->BusInput3.SkipF.rKpTrackLam +
                   Gen2_ref_DWork->DiscreteTimeIntegrator_DSTATE_p) *
    rtb_Switch_jv;

  /* DataTypeConversion: '<S585>/Data Type Conversion1' */
  rtb_Switch2_l = Gen2_ref_B->BusInput3.SkipF.rNum_reserve;

  /* Sum: '<S585>/Sum1' incorporates:
   *  Sum: '<S585>/Sum5'
   */
  rtb_Switch_jv = (Gen2_ref_B->sf_MATLABFunction_n.y + rtb_Switch_fi) +
    rtb_Switch2_l;

  /* MinMax: '<S585>/MinMax' */
  if ((Gen2_ref_B->BusInput.iN_Skip_Ext >= rtb_Switch_jv) || rtIsNaN
      (rtb_Switch_jv)) {
    rtb_Switch_jv = Gen2_ref_B->BusInput.iN_Skip_Ext;
  }

  /* End of MinMax: '<S585>/MinMax' */

  /* Switch: '<S591>/Switch2' incorporates:
   *  Constant: '<S585>/Constant8'
   *  Constant: '<S585>/Constant9'
   *  RelationalOperator: '<S591>/LowerRelop1'
   *  RelationalOperator: '<S591>/UpperRelop'
   *  Sum: '<S585>/Sum8'
   *  Switch: '<S591>/Switch'
   */
  if (rtb_Switch_jv > Gen2_ref_B->BusInput3.eng.rNum_Cyl_Eng - 1.0) {
    rtb_Switch2_ba = Gen2_ref_B->BusInput3.eng.rNum_Cyl_Eng - 1.0;
  } else if (rtb_Switch_jv < 0.0) {
    /* Switch: '<S591>/Switch' incorporates:
     *  Constant: '<S585>/Constant8'
     */
    rtb_Switch2_ba = 0.0;
  } else {
    rtb_Switch2_ba = rtb_Switch_jv;
  }

  /* End of Switch: '<S591>/Switch2' */

  /* Sum: '<S585>/Sum4' */
  rtb_Switch2_n5 = Gen2_ref_B->BusInput3.eng.rNum_Cyl_Eng - rtb_Switch2_ba;

  /* Switch: '<S590>/Switch2' incorporates:
   *  RelationalOperator: '<S590>/LowerRelop1'
   *  RelationalOperator: '<S590>/UpperRelop'
   *  Switch: '<S590>/Switch'
   */
  if (rtb_Switch2_n5 > Gen2_ref_B->BusInput3.eng.rNum_Cyl_Eng) {
    rtb_Switch2_n5 = Gen2_ref_B->BusInput3.eng.rNum_Cyl_Eng;
  } else if (rtb_Switch2_n5 < 1.0) {
    /* Switch: '<S590>/Switch' */
    rtb_Switch2_n5 = 1.0;
  }

  /* End of Switch: '<S590>/Switch2' */

  /* Outputs for Atomic SubSystem: '<S585>/Filter' */
  /* Product: '<S585>/Divide1' */
  Gen2_ref_Filter3(Gen2_ref_B->BusInput3.eng.rNum_Cyl_Eng / rtb_Switch2_n5,
                   Gen2_ref_B->BusInput3.SkipF.rTiF_stat, 1.0, rtb_bResetBdc,
                   &Gen2_ref_B->Filter_n, &Gen2_ref_DWork->Filter_n, inst);

  /* End of Outputs for SubSystem: '<S585>/Filter' */

  /* Switch: '<S8>/Switch2' incorporates:
   *  Constant: '<S8>/Constant2'
   */
  if (Gen2_ref_B->BusInput3.SkipF.bSF_ON) {
    rtb_Divide5_h = Gen2_ref_B->Filter_n.Switch;
  } else {
    rtb_Divide5_h = 1.0;
  }

  /* End of Switch: '<S8>/Switch2' */

  /* MinMax: '<S775>/MinMax' */
  if ((!(rtb_Divide5_h >= Gen2_ref_B->BusInput.tLEANOXin.rHiCtr_Leanox_Corr)) &&
      rtb_bCBV_min) {
    /* MinMax: '<S459>/MinMax' */
    rtb_Divide5_h = Gen2_ref_B->BusInput.tLEANOXin.rHiCtr_Leanox_Corr;
  }

  rtb_Switch2_l = rtb_Divide5_h;

  /* Product: '<S775>/Divide5' incorporates:
   *  Delay: '<S15>/Resettable Delay'
   *  Sum: '<S775>/Add9'
   */
  rtb_Divide6_n = ((rtb_Divide6_n + rtb_Switch1_k) +
                   Gen2_ref_DWork->ResettableDelay_DSTATE) * rtb_Switch2_l;

  /* DataTypeConversion: '<S775>/Data Type Conversion' */
  rtb_Switch2_l = Gen2_ref_B->BusInput.tLEANOXin.rLEANOXoffset;

  /* Sum: '<S432>/Sum' incorporates:
   *  Gain: '<S432>/pa2mbar'
   *  Gain: '<S775>/mbar2pa'
   *  Sum: '<S775>/Add1'
   */
  rtb_Divide6_n = (rtb_Divide6_n + rtb_Switch2_l) * 100.0 * 0.01 +
    Gen2_ref_B->BusInput3.leanox.rPr_Offset_Island;

  /* Switch: '<S759>/Switch2' incorporates:
   *  RelationalOperator: '<S759>/LowerRelop1'
   */
  if (!(rtb_Divide6_n > rtb_mbar2pa_g)) {
    /* Gain: '<S432>/bar2mbar2' */
    rtb_mbar2pa_g = 1000.0 * Gen2_ref_B->BusInput3.traj.rPr_p2s_min;

    /* Switch: '<S759>/Switch' incorporates:
     *  RelationalOperator: '<S759>/UpperRelop'
     */
    if (!(rtb_Divide6_n < rtb_mbar2pa_g)) {
      rtb_mbar2pa_g = rtb_Divide6_n;
    }

    /* End of Switch: '<S759>/Switch' */
  }

  /* End of Switch: '<S759>/Switch2' */

  /* Gain: '<S432>/mbar2pa' */
  rtb_mbar2pa_g *= 100.0;

  /* Sum: '<S760>/Sum1' incorporates:
   *  Constant: '<S760>/Constant1'
   *  DiscreteIntegrator: '<S760>/Discrete-Time Integrator'
   *  Product: '<S760>/Product'
   *  Product: '<S760>/Product1'
   *  Sum: '<S760>/Sum'
   */
  rtb_Switch2_l = (1.0 - Gen2_ref_DWork->DiscreteTimeIntegrator_DSTATE_h) *
    Gen2_ref_B->p2sfilt_l.Switch +
    Gen2_ref_DWork->DiscreteTimeIntegrator_DSTATE_h * rtb_mbar2pa_g;

  /* Switch: '<Root>/BDC_traj3' */
  if (rtb_LogicalOperator) {
    rtb_Divide_kt = rtb_Pa2bar_o;
  } else {
    rtb_Divide_kt = rtb_Switch2_l;
  }

  /* End of Switch: '<Root>/BDC_traj3' */

  /* Sum: '<S307>/Sum3' incorporates:
   *  Gain: '<S307>/Gain'
   *  Gain: '<S307>/Gain1'
   */
  rtb_Product1_b = 1.0E-5 * rtb_Divide_kt - 1.0E-5 * rtb_p2s;

  /* RelationalOperator: '<S307>/Relational Operator' incorporates:
   *  Abs: '<S307>/Abs'
   */
  rtb_LogicalOperator2_e = (fabs(rtb_Product1_b) >
    Gen2_ref_B->BusInput3.fdc.rThrshSwTransFilt);

  /* DiscreteIntegrator: '<S307>/Discrete-Time Integrator' */
  if (rtb_LogicalOperator2_e || (Gen2_ref_DWork->DiscreteTimeIntegrator_PrevRe_p
       != 0)) {
    Gen2_ref_DWork->DiscreteTimeIntegrator_DSTATE_d = 0.0;
  }

  if (Gen2_ref_DWork->DiscreteTimeIntegrator_DSTATE_d >= 1.0) {
    Gen2_ref_DWork->DiscreteTimeIntegrator_DSTATE_d = 1.0;
  } else if (Gen2_ref_DWork->DiscreteTimeIntegrator_DSTATE_d <= 0.0) {
    Gen2_ref_DWork->DiscreteTimeIntegrator_DSTATE_d = 0.0;
  }

  /* DataTypeConversion: '<S4>/Data Type Conversion2' */
  rtb_Product1_b = Gen2_ref_B->BusInput.tPr.rp1LP;

  /* Gain: '<S4>/bar2Pa' */
  rtb_p1LP = 100000.0 * rtb_Product1_b;

  /* MATLAB Function: '<S305>/FILTER no delay' */
  Gen2_ref_FILTERnodelay(rtb_p1LP, Gen2_ref_B->BusInput3.fdc.TiF_Pr_p1,
    Gen2_ref_B->BusInput3.eng.Ts, rtb_bResetBdc, &Gen2_ref_B->sf_FILTERnodelay,
    &Gen2_ref_DWork->sf_FILTERnodelay, inst);

  /* DataTypeConversion: '<S4>/Data Type Conversion3' */
  rtb_Product1_b = Gen2_ref_B->BusInput.tPr.rp1HP;

  /* Gain: '<S4>/bar2Pa1' */
  rtb_p1HP = 100000.0 * rtb_Product1_b;

  /* MATLAB Function: '<S305>/FILTER no delay1' */
  Gen2_ref_FILTERnodelay(rtb_p1HP, Gen2_ref_B->BusInput3.fdc.TiF_Pr_p2_LP,
    Gen2_ref_B->BusInput3.eng.Ts, rtb_bResetBdc, &Gen2_ref_B->sf_FILTERnodelay1,
    &Gen2_ref_DWork->sf_FILTERnodelay1, inst);

  /* DataTypeConversion: '<S4>/Data Type Conversion4' */
  rtb_Product1_b = Gen2_ref_B->BusInput.tPr.rp2HP;

  /* Gain: '<S4>/bar2Pa2' */
  rtb_p2HP = 100000.0 * rtb_Product1_b;

  /* MATLAB Function: '<S305>/FILTER no delay2' */
  Gen2_ref_FILTERnodelay(rtb_p2HP, Gen2_ref_B->BusInput3.fdc.TiF_Pr_p2_HP,
    Gen2_ref_B->BusInput3.eng.Ts, rtb_bResetBdc, &Gen2_ref_B->sf_FILTERnodelay2,
    &Gen2_ref_DWork->sf_FILTERnodelay2, inst);

  /* MATLAB Function: '<S305>/FILTER no delay3' */
  Gen2_ref_FILTERnodelay(rtb_p2s, Gen2_ref_B->BusInput3.fdc.TiF_Pr_p2s,
    Gen2_ref_B->BusInput3.eng.Ts, rtb_bResetBdc, &Gen2_ref_B->sf_FILTERnodelay3,
    &Gen2_ref_DWork->sf_FILTERnodelay3, inst);

  /* Outputs for Atomic SubSystem: '<S306>/2nd Order Filter' */
  Gen2_ref_undOrderFilter(rtb_p1LP,
    Gen2_ref_B->BusInput3.fdc.r2ndOrdFiltOmegaPressure,
    Gen2_ref_B->BusInput3.fdc.r2ndOrdFiltDPressure, rtb_bResetBdc,
    &Gen2_ref_B->undOrderFilter, &Gen2_ref_DWork->undOrderFilter, inst);

  /* End of Outputs for SubSystem: '<S306>/2nd Order Filter' */

  /* Outputs for Atomic SubSystem: '<S306>/2nd Order Filter1' */
  Gen2_ref_undOrderFilter(rtb_p1HP,
    Gen2_ref_B->BusInput3.fdc.r2ndOrdFiltOmegaPressure,
    Gen2_ref_B->BusInput3.fdc.r2ndOrdFiltDPressure, rtb_bResetBdc,
    &Gen2_ref_B->undOrderFilter1, &Gen2_ref_DWork->undOrderFilter1, inst);
```
